# B&R Automation Studio project TD52 (part 63)

```c
  for (i = 0; i < 13; i++) {
    rtb_y_map_new[i] = Gen2_ref_DWork->y_map[i];
  }

  /* End of MATLAB Function: '<S716>/MATLAB Function' */

  /* Switch: '<S636>/Switch6' incorporates:
   *  Constant: '<S636>/Constant2'
   *  Logic: '<S636>/Logical Operator2'
   */
  if (Gen2_ref_B->BusInput3.SpeedCtrl.bKF_GS_xdist1 &&
      Gen2_ref_B->BusInput3.SpeedCtrl.bKF_act) {
    /* Gain: '<S636>/Gain2' */
    rtb_Gain1_o = rtb_Gain3;

    /* S-Function (sfix_look1_dyn): '<S636>/gain scheduling x_dist1' */
    /* Dynamic Look-Up Table Block: '<S636>/gain scheduling x_dist1'
     * Input0  Data Type:  Floating Point real_T
     * Input1  Data Type:  Floating Point real_T
     * Input2  Data Type:  Floating Point real_T
     * Output0 Data Type:  Floating Point real_T
     * Lookup Method: Linear_Endpoint
     *
     */
    LookUp_real_T_real_T( &(rtb_gainschedulingx_dist1), &rtb_y_map_new[0],
                         rtb_Gain1_o,
                         &Gen2_ref_B->BusInput3.SpeedCtrl.refPoint_KF_x_dist1_x
                         [0], 12U, inst);
    rtb_Gain1_o = rtb_gainschedulingx_dist1;
  } else {
    rtb_Gain1_o = 0.0;
  }

  /* SignalConversion generated from: '<S627>/ SFunction ' incorporates:
   *  MATLAB Function: '<S431>/LQR Controller 3states'
   *  Sum: '<S641>/Sum2'
   *  Sum: '<S641>/Sum6'
   */
  rtb_TmpSignalConversionAtSFun_g[0] = rtb_Sum1_l;
  rtb_TmpSignalConversionAtSFun_g[1] = rtb_Sum2_a_tmp;
  rtb_TmpSignalConversionAtSFun_g[2] = rtb_Sum6_o_tmp;

  /* SignalConversion generated from: '<S627>/ SFunction ' incorporates:
   *  MATLAB Function: '<S431>/LQR Controller 3states'
   */
  rtb_Divide_ab[0] = rtb_Sum2_a_tmp;
  rtb_Divide_ab[1] = rtb_Sum6_o_tmp;
  rtb_Divide_ab[2] = rtb_Switch2_oou;
  rtb_Divide_ab[3] = rtb_Sum3_o;

  /* SignalConversion generated from: '<S627>/ SFunction ' incorporates:
   *  Gain: '<S431>/Gain1'
   *  MATLAB Function: '<S431>/LQR Controller 3states'
   */
  rtb_TmpSignalConversionAtSFun_p[0] = rtb_Gain1_f_tmp;
  rtb_TmpSignalConversionAtSFun_p[1] = rtb_Gain3;
  rtb_TmpSignalConversionAtSFun_p[2] = Gen2_ref_B->Filter_bd.Switch;

  /* SignalConversion generated from: '<S627>/ SFunction ' incorporates:
   *  Constant: '<S431>/Nskip_min'
   *  MATLAB Function: '<S431>/LQR Controller 3states'
   */
  rtb_Divide3_e[0] = Gen2_ref_B->BusInput3.traj.rPr_p2s_min;
  rtb_Divide3_e[1] = rtb_Switch1_k;
  rtb_Divide3_e[2] = Gen2_ref_B->BusInput3.SpeedCtrl.rDeltaZZP_min_iLQR;
  rtb_Divide3_e[3] = 0.0;

  /* SignalConversion generated from: '<S627>/ SFunction ' incorporates:
   *  MATLAB Function: '<S431>/LQR Controller 3states'
   */
  rtb_Divide3_i0[0] = Gen2_ref_B->BusInput3.traj.rPr_p2s_max;
  rtb_Divide3_i0[1] = rtb_Switch2_n5;
  rtb_Divide3_i0[2] = Gen2_ref_B->BusInput3.SpeedCtrl.rDeltaZZP_max_iLQR;
  rtb_Divide3_i0[3] = rtb_Switch9_k;

  /* SignalConversion generated from: '<S627>/ SFunction ' incorporates:
   *  Constant: '<S639>/Constant'
   *  DataTypeConversion: '<S639>/Data Type Conversion'
   *  DataTypeConversion: '<S639>/Data Type Conversion1'
   *  MATLAB Function: '<S431>/LQR Controller 3states'
   *  Product: '<S639>/Product'
   */
  rtb_TmpSignalConversionAtSFunct[0] =
    Gen2_ref_B->BusInput3.SpeedCtrl.iNiter_iLQR;
  rtb_TmpSignalConversionAtSFunct[1] = rtb_Product1_b4;
  rtb_TmpSignalConversionAtSFunct[2] = Gen2_ref_B->BusInput3.eng.Ts;
  rtb_TmpSignalConversionAtSFunct[3] = Gen2_ref_B->BusInput3.eng.rJ_Eng *
    Gen2_ref_B->BusInput3.SpeedCtrl.rFactInertiaLQR;
  rtb_TmpSignalConversionAtSFunct[4] = rtb_Product_o;
  rtb_TmpSignalConversionAtSFunct[5] = rtb_Switch_czo;
  rtb_TmpSignalConversionAtSFunct[6] = rtb_Sum2_kg;
  rtb_TmpSignalConversionAtSFunct[7] =
    Gen2_ref_B->BusInput3.SpeedCtrl.rK_it2_iLQR;
  rtb_TmpSignalConversionAtSFunct[8] = rtb_Sum1_idx_2;
  rtb_TmpSignalConversionAtSFunct[9] = rtb_kappa0;
  rtb_TmpSignalConversionAtSFunct[10] =
    Gen2_ref_B->BusInput3.SpeedCtrl.rK_slope_iLQR;
  rtb_TmpSignalConversionAtSFunct[11] =
    Gen2_ref_B->BusInput3.SpeedCtrl.rK_skip_iLQR;
  rtb_TmpSignalConversionAtSFunct[12] = Gen2_ref_B->BusInput3.eng.rNum_Cyl_Eng;
  rtb_TmpSignalConversionAtSFunct[13] =
    Gen2_ref_B->BusInput3.SpeedCtrl.rN_DB_Lambda_act;
  rtb_TmpSignalConversionAtSFunct[14] = 1.0;
  rtb_TmpSignalConversionAtSFunct[15] =
    Gen2_ref_B->BusInput3.SpeedCtrl.iNiterRediLQR;
  rtb_TmpSignalConversionAtSFunct[16] = rtb_Product1_fu;
  rtb_TmpSignalConversionAtSFunct[17] = Gen2_ref_B->BusInput3.eng.rP_Nom;
  rtb_TmpSignalConversionAtSFunct[18] = Gen2_ref_B->BusInput3.eng.rN_Nom;
  rtb_TmpSignalConversionAtSFunct[19] = Gen2_ref_B->BusInput3.traj.rPr_p2s_max;
  rtb_TmpSignalConversionAtSFunct[20] = Gen2_ref_B->BusInput3.LamLim.rLam_max;
  rtb_TmpSignalConversionAtSFunct[21] = rtb_Divide3_g;

  /* MATLAB Function: '<S431>/LQR Controller 3states' incorporates:
   *  DataTypeConversion: '<S639>/Data Type Conversion'
   *  DataTypeConversion: '<S639>/Data Type Conversion1'
   *  Delay: '<S431>/Delay'
   *  Gain: '<S431>/Gain1'
   *  Logic: '<S636>/Logical Operator1'
   *  SignalConversion generated from: '<S627>/ SFunction '
   *  Sum: '<S641>/Sum2'
   *  Sum: '<S641>/Sum6'
   *  Switch: '<S636>/Switch7'
   */
  rtb_Switch2_l = rtb_Gain1_f_tmp;
  y_map_tmp = rtb_Gain3;
  y_map_tmp_0 = Gen2_ref_B->Filter_bd.Switch;
  Gen2_ref_diag(&rtb_Product_m[0], R_2inp, inst);
  Gen2_ref_diag_i(rtb_Product_m, R, inst);
  Gen2_ref_diag_i2(rtb_Switch1_cl, Q, inst);
  for (i = 0; i < 12; i++) {
    rtb_K_LQR[i] = 0.0;
    K_2inp_aug[i] = 0.0;
  }

  delta_y = rt_roundd_snf(rtb_Product1_b4 / Gen2_ref_B->BusInput3.eng.Ts, inst);
  if (delta_y < 32768.0) {
    if (delta_y >= -32768.0) {
      Npred = (int16_T)delta_y;
    } else {
      Npred = MIN_int16_T;
    }
  } else {
    Npred = MAX_int16_T;
  }

  rtb_Product1_b4 = Gen2_ref_B->BusInput3.SpeedCtrl.rN_DB_Lambda_act *
    3.1415926535897931 / 30.0;
  rtb_TmpSignalConversionAtLoo_ht[1] = Gen2_ref_B->BusInput3.eng.rNum_Cyl_Eng;
  if (1.0 < rtb_TmpSignalConversionAtLoo_ht[1]) {
    delta_y = rtb_TmpSignalConversionAtLoo_ht[1];
  } else {
    delta_y = 1.0;
  }

  rtb_Sum2_kg = (1.0 - rtb_Divide3_g / delta_y) * rtb_Product_o;
  Gen2_ref_diag_i2(Gen2_ref_B->BusInput3.SpeedCtrl.rBd_KF, B_d, inst);
  rtb_Switch1_cl[0] = 0.0;
  rtb_Switch1_cl[1] = 0.0;
  rtb_Switch1_cl[2] = 0.0;
  Gen2_ref_diag_i2(Gen2_ref_B->BusInput3.SpeedCtrl.rR_KF, R_KF, inst);
  if (Gen2_ref_B->BusInput3.SpeedCtrl.bKF_x_dist1_AdaptON &&
      Gen2_ref_B->BusInput3.SpeedCtrl.bKF_GS_xdist1 &&
      Gen2_ref_B->TON_j.LogicalOperator3) {
    Gen2_ref_DWork->x_KF[0] = rtb_Gain1_f_tmp;
    Gen2_ref_DWork->x_KF[3] = 0.0;
    Gen2_ref_DWork->x_KF[1] = rtb_Gain3;
    Gen2_ref_DWork->x_KF[4] = 0.0;
    Gen2_ref_DWork->x_KF[2] = Gen2_ref_B->Filter_bd.Switch;
    Gen2_ref_DWork->x_KF[5] = 0.0;
  }

  if ((!Gen2_ref_DWork->P_not_empty) || rtb_bResetHlci) {
    for (i = 0; i < 9; i++) {
      Gen2_ref_DWork->P[i] = 0.0;
    }

    Gen2_ref_DWork->P_not_empty = true;
    for (i = 0; i < 36; i++) {
      Gen2_ref_DWork->P_2inp_aug[i] = 0.0;
    }

    for (i = 0; i < 100; i++) {
      Gen2_ref_DWork->u2_past[i] = rtb_Sum6_o_tmp;
    }

    Gen2_ref_DWork->count = 1.0;
    Gen2_ref_DWork->red_comp = false;
    rtb_Product_m[0] = rtb_Sum2_a_tmp;
    rtb_Product_m[1] = rtb_Sum6_o_tmp;
    rtb_Product_m[2] = rtb_Switch2_oou;
    rtb_Product_m[3] = rtb_Sum3_o;
    Gen2_ref_DWork->x_KF[0] = rtb_Gain1_f_tmp;
    Gen2_ref_DWork->x_KF[3] = 0.0;
    Gen2_ref_DWork->x_KF[1] = rtb_Gain3;
    Gen2_ref_DWork->x_KF[4] = 0.0;
    Gen2_ref_DWork->x_KF[2] = Gen2_ref_B->Filter_bd.Switch;
    Gen2_ref_DWork->x_KF[5] = 0.0;
    for (i = 0; i < 36; i++) {
      Gen2_ref_DWork->P_KF[i] = c[i];
    }

    for (i = 0; i < 18; i++) {
      rtb_K_KF_out[i] = 0.0;
    }

    rtb_err_KF[0] = 0.0;
    rtb_x_KF_out_idx_0 = rtb_Gain1_f_tmp;
    rtb_x_sp_KF_idx_0 = rtb_Sum1_l;
    rtb_err_KF[1] = 0.0;
    rtb_x_KF_out_idx_1 = rtb_Gain3;
    rtb_x_sp_KF_idx_1 = rtb_Sum2_a_tmp;
    rtb_err_KF[2] = 0.0;
    rtb_x_KF_out_idx_2 = Gen2_ref_B->Filter_bd.Switch;
    rtb_x_sp_KF_idx_2 = rtb_Sum6_o_tmp;
    rtb_u_sp_KF[0] = rtb_Sum2_a_tmp;
    rtb_u_sp_KF[1] = rtb_Sum6_o_tmp;
    Gen2_ref_state_space_d(rtb_TmpSignalConversionAtSFun_g,
      rtb_TmpSignalConversionAtSFunct, rtb_Product_o, rtb_Phi_OUT, rtb_H_OUT,
      Hd_obs, inst);
    for (i = 0; i < 3; i++) {
      rtb_err_cont[i] = 0.0;
      Phi_aug_tmp_0 = i << 2;
      K_2inp_aug[Phi_aug_tmp_0] = rtb_H_OUT[i];
      K_2inp_aug[Phi_aug_tmp_0 + 1] = rtb_H_OUT[i + 3];
      K_2inp_aug[Phi_aug_tmp_0 + 2] = rtb_H_OUT[i + 6];
      K_2inp_aug[Phi_aug_tmp_0 + 3] = rtb_H_OUT[i + 9];
    }

    for (i = 0; i < 4; i++) {
      for (Phi_aug_tmp = 0; Phi_aug_tmp < 3; Phi_aug_tmp++) {
        Phi_aug_tmp_0 = (Phi_aug_tmp << 2) + i;
        rtb_H_OUT_0[Phi_aug_tmp_0] = 0.0;
        rtb_H_OUT_0[Phi_aug_tmp_0] += Gen2_ref_DWork->P[3 * Phi_aug_tmp] *
          K_2inp_aug[i];
        rtb_H_OUT_0[Phi_aug_tmp_0] += Gen2_ref_DWork->P[3 * Phi_aug_tmp + 1] *
          K_2inp_aug[i + 4];
        rtb_H_OUT_0[Phi_aug_tmp_0] += Gen2_ref_DWork->P[3 * Phi_aug_tmp + 2] *
          K_2inp_aug[i + 8];
      }

      for (Phi_aug_tmp = 0; Phi_aug_tmp < 4; Phi_aug_tmp++) {
        rtb_H_OUT_tmp = (Phi_aug_tmp << 2) + i;
        R_0[rtb_H_OUT_tmp] = -(((rtb_H_OUT[3 * Phi_aug_tmp + 1] * rtb_H_OUT_0[i
          + 4] + rtb_H_OUT[3 * Phi_aug_tmp] * rtb_H_OUT_0[i]) + rtb_H_OUT[3 *
          Phi_aug_tmp + 2] * rtb_H_OUT_0[i + 8]) + R[rtb_H_OUT_tmp]);
      }
    }

    Gen2_ref_mldivide(R_0, K_2inp_aug, rtb_K_LQR_0, inst);
    for (i = 0; i < 4; i++) {
      for (Phi_aug_tmp = 0; Phi_aug_tmp < 3; Phi_aug_tmp++) {
        rtb_H_OUT_tmp = (Phi_aug_tmp << 2) + i;
        tmp[rtb_H_OUT_tmp] = 0.0;
        tmp[rtb_H_OUT_tmp] += Gen2_ref_DWork->P[3 * Phi_aug_tmp] * rtb_K_LQR_0[i];
        tmp[rtb_H_OUT_tmp] += Gen2_ref_DWork->P[3 * Phi_aug_tmp + 1] *
          rtb_K_LQR_0[i + 4];
        tmp[rtb_H_OUT_tmp] += Gen2_ref_DWork->P[3 * Phi_aug_tmp + 2] *
          rtb_K_LQR_0[i + 8];
      }

      for (Phi_aug_tmp = 0; Phi_aug_tmp < 3; Phi_aug_tmp++) {
        Phi_aug_tmp_0 = (Phi_aug_tmp << 2) + i;
        rtb_K_LQR[Phi_aug_tmp_0] = 0.0;
        rtb_K_LQR[Phi_aug_tmp_0] += rtb_Phi_OUT[3 * Phi_aug_tmp] * tmp[i];
        rtb_K_LQR[Phi_aug_tmp_0] += rtb_Phi_OUT[3 * Phi_aug_tmp + 1] * tmp[i + 4];
        rtb_K_LQR[Phi_aug_tmp_0] += rtb_Phi_OUT[3 * Phi_aug_tmp + 2] * tmp[i + 8];
      }
    }
  } else {
    if (Gen2_ref_DWork->red_comp) {
      rtb_Product1_fu = Gen2_ref_B->BusInput3.SpeedCtrl.iNiterRediLQR;
    } else {
      rtb_Product1_fu = Gen2_ref_B->BusInput3.SpeedCtrl.iNiter_iLQR;
    }

    Gen2_ref_state_space_d(rtb_TmpSignalConversionAtSFun_p,
      rtb_TmpSignalConversionAtSFunct, rtb_Product_o, rtb_Phi_OUT, rtb_H_OUT,
      Hd_obs, inst);
    if (Gen2_ref_B->BusInput3.SpeedCtrl.bKF_KeNskip_Obs) {
      Gen2_ref_state_space_d(rtb_TmpSignalConversionAtSFun_p,
        rtb_TmpSignalConversionAtSFunct, rtb_Sum2_kg, Phi_obs, H_aug, Hd_obs, inst);
    } else {
      Gen2_ref_state_space_d(rtb_TmpSignalConversionAtSFun_p,
        rtb_TmpSignalConversionAtSFunct, rtb_Product_o, Phi_obs, H_aug, Hd_obs, inst);
    }

    if (Gen2_ref_B->BusInput3.SpeedCtrl.bKF_use_Pg) {
      rtb_Sum4_g = rtb_Divide3_ep;
    } else {
      rtb_Sum4_g = rtb_Divide_i1;
    }

    if (Gen2_ref_B->BusInput3.SpeedCtrl.bKF_calc ||
        Gen2_ref_B->BusInput3.SpeedCtrl.bKF_act ||
        Gen2_ref_B->BusInput3.SpeedCtrl.bKF_use_states) {
      rtb_Switch_n = Gen2_ref_B->BusInput3.eng.Ts;
      for (i = 0; i < 3; i++) {
        Phi_aug[6 * i] = Phi_obs[3 * i];
        Phi_aug_tmp_0 = (i + 3) * 6;
        Phi_aug[Phi_aug_tmp_0] = B_d[3 * i] * rtb_Switch_n;
        Phi_aug_tmp = 3 * i + 1;
        Phi_aug[6 * i + 1] = Phi_obs[Phi_aug_tmp];
        Phi_aug[Phi_aug_tmp_0 + 1] = B_d[Phi_aug_tmp] * rtb_Switch_n;
        Phi_aug_tmp = 3 * i + 2;
        Phi_aug[6 * i + 2] = Phi_obs[Phi_aug_tmp];
        Phi_aug[Phi_aug_tmp_0 + 2] = B_d[Phi_aug_tmp] * rtb_Switch_n;
      }

      for (i = 0; i < 6; i++) {
        Phi_aug[6 * i + 3] = b[3 * i];
        Phi_aug[6 * i + 4] = b[3 * i + 1];
        Phi_aug[6 * i + 5] = b[3 * i + 2];
      }

      rtb_Sum5_iu = Gen2_ref_B->BusInput3.eng.rNum_Cyl_Eng;
      if (Gen2_ref_B->BusInput3.eng.rNum_Cyl_Eng < 1.0) {
        rtb_Sum5_iu = 1.0;
      }

      rtb_TmpSignalConversionAtSFun_0[0] = (1.0 - rtb_Divide3_g / rtb_Sum5_iu) *
        rtb_Product_o * Gen2_ref_B->BusInput3.eng.Ts * Gen2_ref_DWork->x_KF[1] /
        ((Gen2_ref_DWork->x_KF[2] * rtb_Sum1_idx_2 + 1.0) *
         rtb_TmpSignalConversionAtSFunct[3]);
      rtb_TmpSignalConversionAtSFun_0[1] = Gen2_ref_B->BusInput3.eng.Ts /
        rtb_Switch_czo * (Gen2_ref_DWork->Delay_DSTATE_ba[0] -
                          Gen2_ref_DWork->x_KF[1]);
      rtb_TmpSignalConversionAtSFun_0[2] = Gen2_ref_B->BusInput3.eng.Ts /
        rtb_TmpSignalConversionAtSFunct[6] * (Gen2_ref_DWork->Delay_DSTATE_ba[1]
        - Gen2_ref_DWork->x_KF[2]);
      rtb_TmpSignalConversionAtSFun_0[3] = 0.0;
      Hd_obs_0[0] = Gen2_ref_DWork->x_KF[0];
      Hd_obs_0[3] = 0.0;
      rtb_TmpSignalConversionAtSFun_0[4] = 0.0;
      Hd_obs_0[1] = Gen2_ref_DWork->x_KF[1];
      Hd_obs_0[4] = 0.0;
      rtb_TmpSignalConversionAtSFun_0[5] = 0.0;
      Hd_obs_0[2] = Gen2_ref_DWork->x_KF[2];
      Hd_obs_0[5] = 0.0;
      for (i = 0; i < 6; i++) {
        rtb_TmpSignalConversionAtSFun_1[i] = ((Phi_aug[i + 18] *
          Gen2_ref_DWork->x_KF[3] + Phi_aug[i + 24] * Gen2_ref_DWork->x_KF[4]) +
          Phi_aug[i + 30] * Gen2_ref_DWork->x_KF[5]) +
          (rtb_TmpSignalConversionAtSFun_0[i] + Hd_obs_0[i]);
      }

      Hd_obs_0[0] = Hd_obs[0] * rtb_Sum4_g;
      Hd_obs_0[3] = 0.0 * rtb_Sum4_g;
      Hd_obs_0[1] = Hd_obs[1] * rtb_Sum4_g;
      Hd_obs_0[4] = 0.0 * rtb_Sum4_g;
      Hd_obs_0[2] = Hd_obs[2] * rtb_Sum4_g;
      Hd_obs_0[5] = 0.0 * rtb_Sum4_g;
      rtb_TmpSignalConversionAtSFun_0[0] = B_d[0] * rtb_Gain1_o *
        Gen2_ref_B->BusInput3.eng.Ts;
      for (i = 0; i < 5; i++) {
        rtb_TmpSignalConversionAtSFun_0[i + 1] = 0.0;
      }

      for (i = 0; i < 6; i++) {
        x_[i] = (rtb_TmpSignalConversionAtSFun_1[i] + Hd_obs_0[i]) +
          rtb_TmpSignalConversionAtSFun_0[i];
        for (Phi_aug_tmp = 0; Phi_aug_tmp < 6; Phi_aug_tmp++) {
          Phi_aug_0[Phi_aug_tmp + 6 * i] = 0.0;
        }

        for (rtb_H_OUT_tmp = 0; rtb_H_OUT_tmp < 6; rtb_H_OUT_tmp++) {
          for (Phi_aug_tmp = 0; Phi_aug_tmp < 6; Phi_aug_tmp++) {
            Phi_aug_tmp_0 = 6 * i + Phi_aug_tmp;
            Phi_aug_0[Phi_aug_tmp_0] += Phi_aug[6 * rtb_H_OUT_tmp + Phi_aug_tmp]
              * Gen2_ref_DWork->P_KF[6 * i + rtb_H_OUT_tmp];
          }
        }
      }

      Gen2_ref_diag_i2a(Gen2_ref_B->BusInput3.SpeedCtrl.rQ_KF, Phi_aug_1, inst);
      for (i = 0; i < 6; i++) {
        for (Phi_aug_tmp = 0; Phi_aug_tmp < 6; Phi_aug_tmp++) {
          delta_y = 0.0;
          for (rtb_H_OUT_tmp = 0; rtb_H_OUT_tmp < 6; rtb_H_OUT_tmp++) {
            delta_y += Phi_aug_0[6 * rtb_H_OUT_tmp + i] * Phi_aug[6 *
              rtb_H_OUT_tmp + Phi_aug_tmp];
          }

          Phi_aug_tmp_0 = 6 * Phi_aug_tmp + i;
          P_[Phi_aug_tmp_0] = Phi_aug_1[Phi_aug_tmp_0] + delta_y;
        }
      }

      for (i = 0; i < 18; i++) {
        Phi_obs_tmp[i] = C_aug[i];
        rtb_K_KF_out[i] = d[i];
      }

      for (i = 0; i < 3; i++) {
        for (Phi_aug_tmp = 0; Phi_aug_tmp < 6; Phi_aug_tmp++) {
          k = 3 * Phi_aug_tmp + i;
          Phi_obs_tmp_0[k] = 0.0;
          for (rtb_H_OUT_tmp = 0; rtb_H_OUT_tmp < 6; rtb_H_OUT_tmp++) {
            Phi_obs_tmp_0[k] += (real_T)Phi_obs_tmp[3 * rtb_H_OUT_tmp + i] * P_
              [6 * Phi_aug_tmp + rtb_H_OUT_tmp];
          }
        }

        for (Phi_aug_tmp = 0; Phi_aug_tmp < 3; Phi_aug_tmp++) {
          delta_y = 0.0;
          for (rtb_H_OUT_tmp = 0; rtb_H_OUT_tmp < 6; rtb_H_OUT_tmp++) {
            delta_y += Phi_obs_tmp_0[3 * rtb_H_OUT_tmp + i] * rtb_K_KF_out[6 *
              Phi_aug_tmp + rtb_H_OUT_tmp];
          }

          k = 3 * Phi_aug_tmp + i;
          Phi_obs[k] = R_KF[k] + delta_y;
        }
      }

      if (fabs(Gen2_ref_det(Phi_obs, inst)) <= 2.2204460492503131E-16) {
        for (i = 0; i < 3; i++) {
          for (Phi_aug_tmp = 0; Phi_aug_tmp < 6; Phi_aug_tmp++) {
            k = 3 * Phi_aug_tmp + i;
            Phi_obs_tmp_0[k] = 0.0;
            for (rtb_H_OUT_tmp = 0; rtb_H_OUT_tmp < 6; rtb_H_OUT_tmp++) {
              Phi_obs_tmp_0[k] += (real_T)Phi_obs_tmp[3 * rtb_H_OUT_tmp + i] *
                Gen2_ref_DWork->P_KF[6 * Phi_aug_tmp + rtb_H_OUT_tmp];
            }
          }

          for (Phi_aug_tmp = 0; Phi_aug_tmp < 3; Phi_aug_tmp++) {
            delta_y = 0.0;
            for (rtb_H_OUT_tmp = 0; rtb_H_OUT_tmp < 6; rtb_H_OUT_tmp++) {
              delta_y += Phi_obs_tmp_0[3 * rtb_H_OUT_tmp + i] * rtb_K_KF_out[6 *
                Phi_aug_tmp + rtb_H_OUT_tmp];
            }

            k = 3 * Phi_aug_tmp + i;
            Phi_obs[k] = R_KF[k] + delta_y;
          }
        }
      }

      for (i = 0; i < 3; i++) {
        for (Phi_aug_tmp = 0; Phi_aug_tmp < 6; Phi_aug_tmp++) {
          Phi_aug_tmp_0 = 6 * i + Phi_aug_tmp;
          Phi_obs_tmp_0[Phi_aug_tmp_0] = 0.0;
          for (rtb_H_OUT_tmp = 0; rtb_H_OUT_tmp < 6; rtb_H_OUT_tmp++) {
            Phi_obs_tmp_0[Phi_aug_tmp_0] += P_[6 * rtb_H_OUT_tmp + Phi_aug_tmp] *
              rtb_K_KF_out[6 * i + rtb_H_OUT_tmp];
          }
        }
      }

      Gen2_ref_mrdiv(Phi_obs_tmp_0, Phi_obs, rtb_K_KF_out, inst);
      for (i = 0; i < 6; i++) {
        for (Phi_aug_tmp = 0; Phi_aug_tmp < 3; Phi_aug_tmp++) {
          k = 6 * Phi_aug_tmp + i;
          Phi_obs_tmp_0[k] = 0.0;
          Phi_obs_tmp_0[k] += Phi_obs[3 * Phi_aug_tmp] * rtb_K_KF_out[i];
          Phi_obs_tmp_0[k] += Phi_obs[3 * Phi_aug_tmp + 1] * rtb_K_KF_out[i + 6];
          Phi_obs_tmp_0[k] += Phi_obs[3 * Phi_aug_tmp + 2] * rtb_K_KF_out[i + 12];
        }

        for (Phi_aug_tmp = 0; Phi_aug_tmp < 6; Phi_aug_tmp++) {
          k = 6 * Phi_aug_tmp + i;
          Gen2_ref_DWork->P_KF[k] = P_[k] - ((Phi_obs_tmp_0[i + 6] *
            rtb_K_KF_out[Phi_aug_tmp + 6] + Phi_obs_tmp_0[i] *
            rtb_K_KF_out[Phi_aug_tmp]) + Phi_obs_tmp_0[i + 12] *
            rtb_K_KF_out[Phi_aug_tmp + 12]);
        }
      }

      for (i = 0; i < 3; i++) {
        Phi_obs_tmp_1[i] = 0.0;
        for (Phi_aug_tmp = 0; Phi_aug_tmp < 6; Phi_aug_tmp++) {
          Phi_obs_tmp_1[i] += (real_T)Phi_obs_tmp[3 * Phi_aug_tmp + i] *
            x_[Phi_aug_tmp];
        }

        rtb_err_KF[i] = (((real_T)b_a[i + 3] * rtb_Gain3 + (real_T)b_a[i] *
                          rtb_Gain1_f_tmp) + (real_T)b_a[i + 6] *
                         Gen2_ref_B->Filter_bd.Switch) - Phi_obs_tmp_1[i];
      }

      for (i = 0; i < 6; i++) {
        Gen2_ref_DWork->x_KF[i] = ((rtb_K_KF_out[i + 6] * rtb_err_KF[1] +
          rtb_K_KF_out[i] * rtb_err_KF[0]) + rtb_K_KF_out[i + 12] * rtb_err_KF[2])
          + x_[i];
      }

      rtb_x_KF_out_idx_0 = Gen2_ref_DWork->x_KF[0];
      rtb_Switch1_cl[0] = Gen2_ref_DWork->x_KF[3];
      rtb_x_KF_out_idx_1 = Gen2_ref_DWork->x_KF[1];
      rtb_Switch1_cl[1] = Gen2_ref_DWork->x_KF[4];
      rtb_x_KF_out_idx_2 = Gen2_ref_DWork->x_KF[2];
      rtb_Switch1_cl[2] = Gen2_ref_DWork->x_KF[5];
      if (Gen2_ref_B->BusInput3.SpeedCtrl.bKF_use_states ||
          Gen2_ref_B->BusInput3.SpeedCtrl.bKF_act) {
        rtb_Switch2_l = Gen2_ref_DWork->x_KF[0];
        y_map_tmp = Gen2_ref_DWork->x_KF[1];
        y_map_tmp_0 = Gen2_ref_DWork->x_KF[2];
      }

      rtb_x_sp_KF_idx_0 = rtb_Sum1_l;
      if (Gen2_ref_B->BusInput3.SpeedCtrl.bKF_constr_handling) {
        if (Gen2_ref_B->BusInput3.SpeedCtrl.bKF_Lam_dyn_SP_shift) {
          FILT_IN = Gen2_ref_DWork->x_KF[3] + rtb_Gain1_o;
          rtb_x_sp_KF_idx_2 = ((FILT_IN * rtb_TmpSignalConversionAtSFunct[3] *
                                B_d[0] + rtb_Sum2_kg * rtb_Sum2_a_tmp) -
                               rtb_Divide_i1) / (rtb_Divide_i1 * rtb_Sum1_idx_2
            - rtb_TmpSignalConversionAtSFunct[3] * rtb_Sum1_idx_2 * FILT_IN *
            B_d[0]) + Gen2_ref_DWork->x_KF[5] * rtb_TmpSignalConversionAtSFunct
            [6] * B_d[8];
        } else {
          rtb_x_sp_KF_idx_1 = Gen2_ref_DWork->x_KF[3] + rtb_Gain1_o;
          rtb_x_sp_KF_idx_2 = ((rtb_x_sp_KF_idx_1 *
                                rtb_TmpSignalConversionAtSFunct[3] * B_d[0] +
                                rtb_Sum2_kg * rtb_Sum2_a_tmp) - rtb_Divide_i1) /
            (rtb_Divide_i1 * rtb_Sum1_idx_2 - rtb_TmpSignalConversionAtSFunct[3]
             * rtb_Sum1_idx_2 * rtb_x_sp_KF_idx_1 * B_d[0]);
        }

        if (rtb_x_sp_KF_idx_2 > rtb_Switch2_n5) {
          rtb_x_sp_KF_idx_2 = rtb_Switch2_n5;
        } else if (rtb_x_sp_KF_idx_2 < rtb_Switch1_k) {
          rtb_x_sp_KF_idx_2 = rtb_Switch1_k;
        }

        if (Gen2_ref_B->BusInput3.SpeedCtrl.bKF_p2s_dyn_SP_shift) {
          rtb_x_sp_KF_idx_1 = (rtb_Divide_i1 - (Gen2_ref_DWork->x_KF[3] +
            rtb_Gain1_o) * rtb_TmpSignalConversionAtSFunct[3] * B_d[0]) *
            (rtb_x_sp_KF_idx_2 * rtb_Sum1_idx_2 + 1.0) / rtb_Sum2_kg +
            Gen2_ref_DWork->x_KF[4] * rtb_Switch_czo * B_d[4];
        } else if ((rtb_Divide3_g > 0.0) &&
                   (!Gen2_ref_B->BusInput3.SpeedCtrl.bKF_constr_handlLR)) {
          rtb_x_sp_KF_idx_1 = rtb_Sum2_a_tmp;
        } else {
          rtb_x_sp_KF_idx_1 = (rtb_Divide_i1 - (Gen2_ref_DWork->x_KF[3] +
            rtb_Gain1_o) * rtb_TmpSignalConversionAtSFunct[3] * B_d[0]) *
            (rtb_x_sp_KF_idx_2 * rtb_Sum1_idx_2 + 1.0) / rtb_Sum2_kg;
        }
      } else {
        if (Gen2_ref_B->BusInput3.SpeedCtrl.bKF_p2s_dyn_SP_shift) {
          rtb_x_sp_KF_idx_1 = Gen2_ref_DWork->x_KF[4] * rtb_Switch_czo * B_d[4]
            + rtb_Sum2_a_tmp;
        } else {
          rtb_x_sp_KF_idx_1 = rtb_Sum2_a_tmp;
        }

        if (Gen2_ref_B->BusInput3.SpeedCtrl.bKF_Lam_dyn_SP_shift) {
          rtb_x_sp_KF_idx_2 = (((Gen2_ref_DWork->x_KF[3] + rtb_Gain1_o) *
                                rtb_TmpSignalConversionAtSFunct[3] * B_d[0] +
                                rtb_Sum2_kg * rtb_Sum2_a_tmp) - rtb_Divide_i1) /
            (rtb_Divide_i1 * rtb_Sum1_idx_2 - rtb_TmpSignalConversionAtSFunct[3]
             * rtb_Sum1_idx_2 * (Gen2_ref_DWork->x_KF[3] + rtb_Gain1_o) * B_d[0])
            + Gen2_ref_DWork->x_KF[5] * rtb_TmpSignalConversionAtSFunct[6] *
            B_d[8];
        } else {
          rtb_x_sp_KF_idx_2 = (((Gen2_ref_DWork->x_KF[3] + rtb_Gain1_o) *
                                rtb_TmpSignalConversionAtSFunct[3] * B_d[0] +
                                rtb_Sum2_kg * rtb_Sum2_a_tmp) - rtb_Divide_i1) /
            (rtb_Divide_i1 * rtb_Sum1_idx_2 - rtb_TmpSignalConversionAtSFunct[3]
             * rtb_Sum1_idx_2 * (Gen2_ref_DWork->x_KF[3] + rtb_Gain1_o) * B_d[0]);
        }
      }

      rtb_u_sp_KF[0] = rtb_x_sp_KF_idx_1;
      rtb_u_sp_KF[1] = rtb_x_sp_KF_idx_2;
    } else {
      rtb_err_KF[0] = 0.0;
      rtb_x_KF_out_idx_0 = rtb_Gain1_f_tmp * 0.0;
      rtb_x_sp_KF_idx_0 = 0.0;
      rtb_err_KF[1] = 0.0;
      rtb_x_KF_out_idx_1 = rtb_Gain3 * 0.0;
      rtb_x_sp_KF_idx_1 = 0.0;
      rtb_err_KF[2] = 0.0;
      rtb_x_KF_out_idx_2 = Gen2_ref_B->Filter_bd.Switch * 0.0;
      rtb_x_sp_KF_idx_2 = 0.0;
      rtb_u_sp_KF[0] = 0.0;
      rtb_u_sp_KF[1] = 0.0;
      for (i = 0; i < 18; i++) {
        rtb_K_KF_out[i] = 0.0;
      }
    }

    rtb_err_cont[0] = rtb_Sum1_l - rtb_Switch2_l;
    rtb_err_cont[1] = rtb_Sum2_a_tmp - y_map_tmp;
    rtb_err_cont[2] = rtb_Sum6_o_tmp - y_map_tmp_0;
    if (Gen2_ref_B->BusInput3.SpeedCtrl.bKF_act) {
      rtb_Switch_n = Gen2_ref_B->BusInput3.eng.Ts;
      for (i = 0; i < 3; i++) {
        Phi_aug[6 * i] = rtb_Phi_OUT[3 * i];
        Phi_aug_tmp_0 = (i + 3) * 6;
        Phi_aug[Phi_aug_tmp_0] = B_d[3 * i] * rtb_Switch_n;
        Phi_aug_tmp = 3 * i + 1;
        Phi_aug[6 * i + 1] = rtb_Phi_OUT[Phi_aug_tmp];
        Phi_aug[Phi_aug_tmp_0 + 1] = B_d[Phi_aug_tmp] * rtb_Switch_n;
        Phi_aug_tmp = 3 * i + 2;
        Phi_aug[6 * i + 2] = rtb_Phi_OUT[Phi_aug_tmp];
        Phi_aug[Phi_aug_tmp_0 + 2] = B_d[Phi_aug_tmp] * rtb_Switch_n;
      }

      for (i = 0; i < 6; i++) {
        Phi_aug[6 * i + 3] = b[3 * i];
        Phi_aug[6 * i + 4] = b[3 * i + 1];
        Phi_aug[6 * i + 5] = b[3 * i + 2];
      }

      for (i = 0; i < 2; i++) {
        H_aug[6 * i] = rtb_H_OUT[3 * i];
        H_aug[6 * i + 3] = 0.0;
        H_aug[6 * i + 1] = rtb_H_OUT[3 * i + 1];
        H_aug[6 * i + 4] = 0.0;
        H_aug[6 * i + 2] = rtb_H_OUT[3 * i + 2];
        H_aug[6 * i + 5] = 0.0;
      }

      for (i = 0; i < 3; i++) {
        P_[6 * i] = Q[3 * i];
        Phi_aug_tmp_0 = (i + 3) * 6;
        P_[Phi_aug_tmp_0] = 0.0;
        P_[6 * i + 1] = Q[3 * i + 1];
        P_[Phi_aug_tmp_0 + 1] = 0.0;
        P_[6 * i + 2] = Q[3 * i + 2];
        P_[Phi_aug_tmp_0 + 2] = 0.0;
      }

      for (i = 0; i < 6; i++) {
        P_[6 * i + 3] = 0.0;
        P_[6 * i + 4] = 0.0;
        P_[6 * i + 5] = 0.0;
      }

      if (0 <= (int32_T)rtb_Product1_fu - 1) {
        for (i = 0; i < 6; i++) {
          Phi_aug_tmp_0 = i << 1;
          rtb_K_LQR[Phi_aug_tmp_0] = H_aug[i];
          rtb_K_LQR[Phi_aug_tmp_0 + 1] = H_aug[i + 6];
        }
      }

      for (k = 0; k < (int32_T)rtb_Product1_fu; k++) {
        for (i = 0; i < 2; i++) {
          for (Phi_aug_tmp = 0; Phi_aug_tmp < 6; Phi_aug_tmp++) {
            Phi_aug_tmp_0 = (Phi_aug_tmp << 1) + i;
            rtb_K_LQR_0[Phi_aug_tmp_0] = 0.0;
            for (rtb_H_OUT_tmp = 0; rtb_H_OUT_tmp < 6; rtb_H_OUT_tmp++) {
              rtb_K_LQR_0[Phi_aug_tmp_0] += rtb_K_LQR[(rtb_H_OUT_tmp << 1) + i] *
                Gen2_ref_DWork->P_2inp_aug[6 * Phi_aug_tmp + rtb_H_OUT_tmp];
            }
          }

          for (Phi_aug_tmp = 0; Phi_aug_tmp < 2; Phi_aug_tmp++) {
            delta_y = 0.0;
            for (rtb_H_OUT_tmp = 0; rtb_H_OUT_tmp < 6; rtb_H_OUT_tmp++) {
              delta_y += rtb_K_LQR_0[(rtb_H_OUT_tmp << 1) + i] * H_aug[6 *
                Phi_aug_tmp + rtb_H_OUT_tmp];
            }

            rtb_H_OUT_tmp = (Phi_aug_tmp << 1) + i;
            rtb_Product_m[rtb_H_OUT_tmp] = -(R_2inp[rtb_H_OUT_tmp] + delta_y);
          }
        }

        Gen2_ref_mldivide_j(rtb_Product_m, rtb_K_LQR, rtb_K_LQR_0, inst);
        for (i = 0; i < 2; i++) {
          for (Phi_aug_tmp = 0; Phi_aug_tmp < 6; Phi_aug_tmp++) {
            rtb_H_OUT_tmp = (Phi_aug_tmp << 1) + i;
            tmp[rtb_H_OUT_tmp] = 0.0;
            for (Phi_aug_tmp_0 = 0; Phi_aug_tmp_0 < 6; Phi_aug_tmp_0++) {
              tmp[rtb_H_OUT_tmp] += rtb_K_LQR_0[(Phi_aug_tmp_0 << 1) + i] *
                Gen2_ref_DWork->P_2inp_aug[6 * Phi_aug_tmp + Phi_aug_tmp_0];
            }
          }

          for (Phi_aug_tmp = 0; Phi_aug_tmp < 6; Phi_aug_tmp++) {
            Phi_aug_tmp_0 = (Phi_aug_tmp << 1) + i;
            K_2inp_aug[Phi_aug_tmp_0] = 0.0;
            for (rtb_H_OUT_tmp = 0; rtb_H_OUT_tmp < 6; rtb_H_OUT_tmp++) {
              K_2inp_aug[Phi_aug_tmp_0] += tmp[(rtb_H_OUT_tmp << 1) + i] *
                Phi_aug[6 * Phi_aug_tmp + rtb_H_OUT_tmp];
            }
          }
        }

        for (i = 0; i < 6; i++) {
          rtb_H_OUT_0[i] = 0.0;
          Phi_aug_tmp_0 = i << 1;
          rtb_Sum2_kg = K_2inp_aug[Phi_aug_tmp_0];
          rtb_H_OUT_0[i] += rtb_Sum2_kg * R_2inp[0];
          rtb_Switch_czo = K_2inp_aug[Phi_aug_tmp_0 + 1];
          rtb_H_OUT_0[i] += rtb_Switch_czo * R_2inp[1];
          rtb_H_OUT_0[i + 6] = 0.0;
          rtb_H_OUT_0[i + 6] += rtb_Sum2_kg * R_2inp[2];
          rtb_H_OUT_0[i + 6] += rtb_Switch_czo * R_2inp[3];
          for (Phi_aug_tmp = 0; Phi_aug_tmp < 6; Phi_aug_tmp++) {
            rtb_H_OUT_tmp = 6 * Phi_aug_tmp + i;
            P_2inp_aug_tmp[rtb_H_OUT_tmp] = 0.0;
            Phi_aug_tmp_0 = Phi_aug_tmp << 1;
            P_2inp_aug_tmp[rtb_H_OUT_tmp] += K_2inp_aug[Phi_aug_tmp_0] * H_aug[i];
            P_2inp_aug_tmp[rtb_H_OUT_tmp] += K_2inp_aug[Phi_aug_tmp_0 + 1] *
              H_aug[i + 6];
            Phi_aug_0[Phi_aug_tmp + 6 * i] = Phi_aug[rtb_H_OUT_tmp] +
              P_2inp_aug_tmp[rtb_H_OUT_tmp];
          }
        }

        for (i = 0; i < 6; i++) {
          for (Phi_aug_tmp = 0; Phi_aug_tmp < 6; Phi_aug_tmp++) {
            Phi_aug_tmp_0 = 6 * Phi_aug_tmp + i;
            Phi_aug_1[Phi_aug_tmp_0] = 0.0;
            for (rtb_H_OUT_tmp = 0; rtb_H_OUT_tmp < 6; rtb_H_OUT_tmp++) {
              Phi_aug_1[Phi_aug_tmp_0] += Phi_aug_0[6 * rtb_H_OUT_tmp + i] *
                Gen2_ref_DWork->P_2inp_aug[6 * Phi_aug_tmp + rtb_H_OUT_tmp];
            }
          }
        }

        for (i = 0; i < 36; i++) {
          Phi_aug_0[i] = Phi_aug[i] + P_2inp_aug_tmp[i];
        }

        for (i = 0; i < 6; i++) {
          for (Phi_aug_tmp = 0; Phi_aug_tmp < 6; Phi_aug_tmp++) {
            Phi_aug_tmp_0 = Phi_aug_tmp << 1;
            rtb_K_LQR_tmp = 6 * Phi_aug_tmp + i;
            P_2inp_aug_tmp[rtb_K_LQR_tmp] = (K_2inp_aug[Phi_aug_tmp_0 + 1] *
              rtb_H_OUT_0[i + 6] + K_2inp_aug[Phi_aug_tmp_0] * rtb_H_OUT_0[i]) +
              P_[rtb_K_LQR_tmp];
            Phi_aug_2[rtb_K_LQR_tmp] = 0.0;
            for (rtb_H_OUT_tmp = 0; rtb_H_OUT_tmp < 6; rtb_H_OUT_tmp++) {
              Phi_aug_2[rtb_K_LQR_tmp] += Phi_aug_1[6 * rtb_H_OUT_tmp + i] *
                Phi_aug_0[6 * Phi_aug_tmp + rtb_H_OUT_tmp];
            }
          }
        }

        for (i = 0; i < 36; i++) {
          Gen2_ref_DWork->P_2inp_aug[i] = P_2inp_aug_tmp[i] + Phi_aug_2[i];
        }
      }

      for (i = 0; i < 3; i++) {
        Phi_aug_tmp_0 = i << 2;
        rtb_H_OUT_tmp = i << 1;
        rtb_K_LQR[Phi_aug_tmp_0] = K_2inp_aug[rtb_H_OUT_tmp];
        rtb_K_LQR[Phi_aug_tmp_0 + 2] = 0.0;
        rtb_K_LQR[Phi_aug_tmp_0 + 1] = K_2inp_aug[rtb_H_OUT_tmp + 1];
        rtb_K_LQR[Phi_aug_tmp_0 + 3] = 0.0;
        Gen2_ref_DWork->P[3 * i] = Gen2_ref_DWork->P_2inp_aug[6 * i];
        Gen2_ref_DWork->P[3 * i + 1] = Gen2_ref_DWork->P_2inp_aug[6 * i + 1];
        Gen2_ref_DWork->P[3 * i + 2] = Gen2_ref_DWork->P_2inp_aug[6 * i + 2];
      }
    } else {
      if (0 <= (int32_T)rtb_Product1_fu - 1) {
        for (i = 0; i < 3; i++) {
          rtb_H_OUT_tmp = i << 2;
          rtb_H_OUT_0[rtb_H_OUT_tmp] = rtb_H_OUT[i];
          rtb_H_OUT_0[rtb_H_OUT_tmp + 1] = rtb_H_OUT[i + 3];
          rtb_H_OUT_0[rtb_H_OUT_tmp + 2] = rtb_H_OUT[i + 6];
          rtb_H_OUT_0[rtb_H_OUT_tmp + 3] = rtb_H_OUT[i + 9];
        }
      }

      for (k = 0; k < (int32_T)rtb_Product1_fu; k++) {
        for (i = 0; i < 4; i++) {
          for (Phi_aug_tmp = 0; Phi_aug_tmp < 3; Phi_aug_tmp++) {
            rtb_H_OUT_tmp = (Phi_aug_tmp << 2) + i;
            rtb_K_LQR[rtb_H_OUT_tmp] = 0.0;
            rtb_K_LQR[rtb_H_OUT_tmp] += rtb_H_OUT[3 * i] * Gen2_ref_DWork->P[3 *
              Phi_aug_tmp];
            rtb_K_LQR[rtb_H_OUT_tmp] += rtb_H_OUT[3 * i + 1] * Gen2_ref_DWork->
              P[3 * Phi_aug_tmp + 1];
            rtb_K_LQR[rtb_H_OUT_tmp] += rtb_H_OUT[3 * i + 2] * Gen2_ref_DWork->
              P[3 * Phi_aug_tmp + 2];
          }

          for (Phi_aug_tmp = 0; Phi_aug_tmp < 4; Phi_aug_tmp++) {
            rtb_H_OUT_tmp = (Phi_aug_tmp << 2) + i;
            R_0[rtb_H_OUT_tmp] = -(((rtb_H_OUT[3 * Phi_aug_tmp + 1] *
              rtb_K_LQR[i + 4] + rtb_H_OUT[3 * Phi_aug_tmp] * rtb_K_LQR[i]) +
              rtb_H_OUT[3 * Phi_aug_tmp + 2] * rtb_K_LQR[i + 8]) +
              R[rtb_H_OUT_tmp]);
          }
        }

        Gen2_ref_mldivide(R_0, rtb_H_OUT_0, rtb_K_LQR_0, inst);
        for (i = 0; i < 4; i++) {
          for (Phi_aug_tmp = 0; Phi_aug_tmp < 3; Phi_aug_tmp++) {
            rtb_H_OUT_tmp = (Phi_aug_tmp << 2) + i;
            tmp[rtb_H_OUT_tmp] = 0.0;
            tmp[rtb_H_OUT_tmp] += Gen2_ref_DWork->P[3 * Phi_aug_tmp] *
              rtb_K_LQR_0[i];
            tmp[rtb_H_OUT_tmp] += Gen2_ref_DWork->P[3 * Phi_aug_tmp + 1] *
              rtb_K_LQR_0[i + 4];
            tmp[rtb_H_OUT_tmp] += Gen2_ref_DWork->P[3 * Phi_aug_tmp + 2] *
              rtb_K_LQR_0[i + 8];
          }

          for (Phi_aug_tmp = 0; Phi_aug_tmp < 3; Phi_aug_tmp++) {
            Phi_aug_tmp_0 = (Phi_aug_tmp << 2) + i;
            rtb_K_LQR[Phi_aug_tmp_0] = 0.0;
            rtb_K_LQR[Phi_aug_tmp_0] += rtb_Phi_OUT[3 * Phi_aug_tmp] * tmp[i];
            rtb_K_LQR[Phi_aug_tmp_0] += rtb_Phi_OUT[3 * Phi_aug_tmp + 1] * tmp[i
              + 4];
            rtb_K_LQR[Phi_aug_tmp_0] += rtb_Phi_OUT[3 * Phi_aug_tmp + 2] * tmp[i
              + 8];
          }
        }

        for (i = 0; i < 3; i++) {
          for (Phi_aug_tmp = 0; Phi_aug_tmp < 3; Phi_aug_tmp++) {
            rtb_H_OUT_tmp = 3 * Phi_aug_tmp + i;
            R_KF[rtb_H_OUT_tmp] = 0.0;
            Phi_aug_tmp_0 = Phi_aug_tmp << 2;
            R_KF[rtb_H_OUT_tmp] += rtb_K_LQR[Phi_aug_tmp_0] * rtb_H_OUT[i];
            R_KF[rtb_H_OUT_tmp] += rtb_K_LQR[Phi_aug_tmp_0 + 1] * rtb_H_OUT[i +
              3];
            R_KF[rtb_H_OUT_tmp] += rtb_K_LQR[Phi_aug_tmp_0 + 2] * rtb_H_OUT[i +
              6];
            R_KF[rtb_H_OUT_tmp] += rtb_K_LQR[Phi_aug_tmp_0 + 3] * rtb_H_OUT[i +
              9];
          }

          for (Phi_aug_tmp = 0; Phi_aug_tmp < 4; Phi_aug_tmp++) {
            Phi_aug_tmp_0 = 3 * Phi_aug_tmp + i;
            rtb_K_LQR_0[Phi_aug_tmp_0] = 0.0;
            rtb_H_OUT_tmp = i << 2;
            rtb_K_LQR_tmp = Phi_aug_tmp << 2;
            rtb_K_LQR_0[Phi_aug_tmp_0] += rtb_K_LQR[rtb_H_OUT_tmp] *
              R[rtb_K_LQR_tmp];
            rtb_K_LQR_0[Phi_aug_tmp_0] += rtb_K_LQR[rtb_H_OUT_tmp + 1] *
              R[rtb_K_LQR_tmp + 1];
            rtb_K_LQR_0[Phi_aug_tmp_0] += rtb_K_LQR[rtb_H_OUT_tmp + 2] *
              R[rtb_K_LQR_tmp + 2];
            rtb_K_LQR_0[Phi_aug_tmp_0] += rtb_K_LQR[rtb_H_OUT_tmp + 3] *
              R[rtb_K_LQR_tmp + 3];
          }

          Phi_obs[3 * i] = rtb_Phi_OUT[i] + R_KF[i];
          Phi_obs[3 * i + 1] = rtb_Phi_OUT[i + 3] + R_KF[i + 3];
          Phi_obs[3 * i + 2] = rtb_Phi_OUT[i + 6] + R_KF[i + 6];
        }

        for (i = 0; i < 3; i++) {
          for (Phi_aug_tmp = 0; Phi_aug_tmp < 3; Phi_aug_tmp++) {
            rtb_H_OUT_tmp = 3 * Phi_aug_tmp + i;
            rtb_Phi_OUT_0[rtb_H_OUT_tmp] = 0.0;
            rtb_Phi_OUT_0[rtb_H_OUT_tmp] += Gen2_ref_DWork->P[3 * Phi_aug_tmp] *
              Phi_obs[i];
            rtb_Phi_OUT_0[rtb_H_OUT_tmp] += Gen2_ref_DWork->P[3 * Phi_aug_tmp +
              1] * Phi_obs[i + 3];
            rtb_Phi_OUT_0[rtb_H_OUT_tmp] += Gen2_ref_DWork->P[3 * Phi_aug_tmp +
              2] * Phi_obs[i + 6];
          }
        }

        for (i = 0; i < 9; i++) {
          Phi_obs[i] = rtb_Phi_OUT[i] + R_KF[i];
        }

        for (i = 0; i < 3; i++) {
          for (Phi_aug_tmp = 0; Phi_aug_tmp < 3; Phi_aug_tmp++) {
            rtb_H_OUT_tmp = Phi_aug_tmp << 2;
            Phi_aug_tmp_0 = 3 * Phi_aug_tmp + i;
            R_KF[Phi_aug_tmp_0] = (((rtb_K_LQR[rtb_H_OUT_tmp + 1] *
              rtb_K_LQR_0[i + 3] + rtb_K_LQR[rtb_H_OUT_tmp] * rtb_K_LQR_0[i]) +
              rtb_K_LQR[rtb_H_OUT_tmp + 2] * rtb_K_LQR_0[i + 6]) +
              rtb_K_LQR[rtb_H_OUT_tmp + 3] * rtb_K_LQR_0[i + 9]) +
              Q[Phi_aug_tmp_0];
            rtb_Phi_OUT_1[Phi_aug_tmp_0] = 0.0;
            rtb_Phi_OUT_1[Phi_aug_tmp_0] += Phi_obs[3 * Phi_aug_tmp] *
              rtb_Phi_OUT_0[i];
            rtb_Phi_OUT_1[Phi_aug_tmp_0] += Phi_obs[3 * Phi_aug_tmp + 1] *
              rtb_Phi_OUT_0[i + 3];
            rtb_Phi_OUT_1[Phi_aug_tmp_0] += Phi_obs[3 * Phi_aug_tmp + 2] *
              rtb_Phi_OUT_0[i + 6];
          }
        }

        for (i = 0; i < 9; i++) {
          Gen2_ref_DWork->P[i] = R_KF[i] + rtb_Phi_OUT_1[i];
        }
      }
    }

    rtb_TmpSignalConversionAtSFun_0[0] = rtb_x_sp_KF_idx_0;
    rtb_TmpSignalConversionAtSFun_0[3] = 0.0;
    rtb_TmpSignalConversionAtSFun_1[0] = rtb_Switch2_l;
    rtb_TmpSignalConversionAtSFun_1[3] = 0.0;
    rtb_TmpSignalConversionAtSFun_0[1] = rtb_x_sp_KF_idx_1;
    rtb_TmpSignalConversionAtSFun_0[4] = 0.0;
    rtb_TmpSignalConversionAtSFun_1[1] = y_map_tmp;
    rtb_TmpSignalConversionAtSFun_1[4] = 0.0;
    rtb_TmpSignalConversionAtSFun_0[2] = rtb_x_sp_KF_idx_2;
    rtb_TmpSignalConversionAtSFun_0[5] = 0.0;
    rtb_TmpSignalConversionAtSFun_1[2] = y_map_tmp_0;
    rtb_TmpSignalConversionAtSFun_1[5] = 0.0;
    for (i = 0; i < 6; i++) {
      Hd_obs_0[i] = rtb_TmpSignalConversionAtSFun_0[i] -
        rtb_TmpSignalConversionAtSFun_1[i];
    }

    for (i = 0; i < 2; i++) {
      delta_y = 0.0;
      for (Phi_aug_tmp = 0; Phi_aug_tmp < 6; Phi_aug_tmp++) {
        delta_y += K_2inp_aug[(Phi_aug_tmp << 1) + i] * Hd_obs_0[Phi_aug_tmp];
      }

      R_2inp[i] = rtb_u_sp_KF[i] - delta_y;
    }

    R_2inp[2] = 0.0;
    R_2inp[3] = 0.0;
    if (Gen2_ref_B->BusInput3.SpeedCtrl.bKF_act) {
      for (i = 0; i < 4; i++) {
        rtb_Product_m[i] = R_2inp[i];
      }

      for (i = 0; i < 3; i++) {
        Phi_aug_tmp = i << 2;
        k = i << 1;
        H_aug[Phi_aug_tmp] = K_2inp_aug[k];
        H_aug[Phi_aug_tmp + 2] = 0.0;
        H_aug[Phi_aug_tmp + 1] = K_2inp_aug[k + 1];
        H_aug[Phi_aug_tmp + 3] = 0.0;
      }

      R_2inp[0] = rtb_u_sp_KF[0];
      R_2inp[1] = rtb_u_sp_KF[1];
      R_2inp[2] = 0.0;
      R_2inp[3] = 0.0;
      Hd_obs[0] = rtb_x_sp_KF_idx_0;
      Hd_obs[1] = rtb_x_sp_KF_idx_1;
      Hd_obs[2] = rtb_x_sp_KF_idx_2;
    } else {
      for (i = 0; i < 4; i++) {
        rtb_Product_m[i] = rtb_Divide_ab[i] - ((rtb_K_LQR[i + 4] * rtb_err_cont
          [1] + rtb_K_LQR[i] * rtb_err_cont[0]) + rtb_K_LQR[i + 8] *
          rtb_err_cont[2]);
      }

      for (i = 0; i < 12; i++) {
        H_aug[i] = rtb_K_LQR[i];
      }

      R_2inp[0] = rtb_Sum2_a_tmp;
      R_2inp[1] = rtb_Sum6_o_tmp;
      R_2inp[2] = rtb_Switch2_oou;
      R_2inp[3] = rtb_Sum3_o;
      Hd_obs[0] = rtb_Sum1_l;
      Hd_obs[1] = rtb_Sum2_a_tmp;
      Hd_obs[2] = rtb_Sum6_o_tmp;
    }

    for (i = 0; i < 100; i++) {
      u_lambda_past[i] = 0.0;
    }

    for (k = 1; k - 1 < Npred; k++) {
      i = Npred + 1;
      if (Npred + 1 > 32767) {
        i = 32767;
      }

      delta_y = rt_roundd_snf(Gen2_ref_DWork->count - (real_T)i, inst);
      if (delta_y < 32768.0) {
        if (delta_y >= -32768.0) {
          tmp_0 = (int16_T)delta_y;
        } else {
          tmp_0 = MIN_int16_T;
        }
      } else {
        tmp_0 = MAX_int16_T;
      }

      i = tmp_0 + (int16_T)k;
      if (i > 32767) {
        i = 32767;
      } else if (i < -32768) {
        i = -32768;
      }

      if (i < 1) {
        i = Npred + 1;
        if (Npred + 1 > 32767) {
          i = 32767;
        }

        delta_y = rt_roundd_snf((real_T)i - Gen2_ref_DWork->count, inst);
        if (delta_y < 32768.0) {
          if (delta_y >= -32768.0) {
            tmp_0 = (int16_T)delta_y;
          } else {
            tmp_0 = MIN_int16_T;
          }
        } else {
          tmp_0 = MAX_int16_T;
        }

        i = 100 - tmp_0;
        if (delta_y < 32768.0) {
          if (delta_y >= -32768.0) {
            tmp_0 = (int16_T)delta_y;
          } else {
            tmp_0 = MIN_int16_T;
          }
        } else {
          tmp_0 = MAX_int16_T;
        }

        if (100 - tmp_0 > 32767) {
          i = 32767;
        }

        i += (int16_T)k;
        if (i > 32767) {
          i = 32767;
        } else if (i < -32768) {
          i = -32768;
        }

        u_lambda_past[(int16_T)k - 1] = Gen2_ref_DWork->u2_past[i - 1];
      } else {
        i = Npred + 1;
        if (Npred + 1 > 32767) {
          i = 32767;
        }

        delta_y = rt_roundd_snf(Gen2_ref_DWork->count - (real_T)i, inst);
        if (delta_y < 32768.0) {
          if (delta_y >= -32768.0) {
            tmp_0 = (int16_T)delta_y;
          } else {
            tmp_0 = MIN_int16_T;
          }
        } else {
          tmp_0 = MAX_int16_T;
        }

        i = tmp_0 + (int16_T)k;
        if (i > 32767) {
          i = 32767;
        } else if (i < -32768) {
          i = -32768;
        }

        u_lambda_past[(int16_T)k - 1] = Gen2_ref_DWork->u2_past[i - 1];
      }
    }

    rtb_TmpSignalConversionAtSFun_g[0] = rtb_Switch2_l;
    rtb_TmpSignalConversionAtSFun_g[1] = y_map_tmp;
    rtb_TmpSignalConversionAtSFun_g[2] = y_map_tmp_0;
    if (!Gen2_ref_B->BusInput3.SpeedCtrl.bPredFB_usePg) {
      rtb_Divide3_ep = rtb_Divide_i1;
    }

    Gen2_ref_integrate_model(rtb_TmpSignalConversionAtSFun_g, H_aug,
      u_lambda_past, rtb_Divide3_ep, rtb_Switch1_cl, B_d, rtb_Gain1_o, R_2inp,
      Hd_obs, Npred, rtb_Divide3_e, rtb_Divide3_i0,
      rtb_TmpSignalConversionAtSFunct, inst);
    if (rtb_Product1_b4 > 0.5) {
      rtb_Product1_fu = Hd_obs[0] - rtb_TmpSignalConversionAtSFun_g[0];
      if (rtb_Product1_fu > 0.0) {
        u0 = rtb_Product1_fu - rtb_Product1_b4;
        if (u0 >= 0.0) {
          Hd_obs[0] = u0;
        } else {
          Hd_obs[0] = 0.0;
        }
      } else {
        u0 = rtb_Product1_fu + rtb_Product1_b4;
        if (u0 <= 0.0) {
          Hd_obs[0] = u0;
        } else {
          Hd_obs[0] = 0.0;
        }
      }

      rtb_Product_m[1] = R_2inp[1] - (((Hd_obs[1] -
        rtb_TmpSignalConversionAtSFun_g[1]) * H_aug[5] + Hd_obs[0] * H_aug[1]) +
        (Hd_obs[2] - rtb_TmpSignalConversionAtSFun_g[2]) * H_aug[9]);
    } else {
      rtb_Product_m[1] = R_2inp[1] - (((Hd_obs[0] -
        rtb_TmpSignalConversionAtSFun_g[0]) * H_aug[1] + (Hd_obs[1] -
        rtb_TmpSignalConversionAtSFun_g[1]) * H_aug[5]) + (Hd_obs[2] -
        rtb_TmpSignalConversionAtSFun_g[2]) * H_aug[9]);
    }

    rtb_Product1_b4 = rtb_Product_m[0];
    if (rtb_Product_m[0] > Gen2_ref_B->BusInput3.traj.rPr_p2s_max) {
      rtb_Product1_b4 = Gen2_ref_B->BusInput3.traj.rPr_p2s_max;
    } else if (rtb_Product_m[0] < Gen2_ref_B->BusInput3.traj.rPr_p2s_min) {
      rtb_Product1_b4 = Gen2_ref_B->BusInput3.traj.rPr_p2s_min;
    }

    rtb_Product_m[0] = rtb_Product1_b4;
    rtb_Product1_b4 = rtb_Product_m[1];
    if (rtb_Product_m[1] > rtb_Switch2_n5) {
      rtb_Product1_b4 = rtb_Switch2_n5;
    } else if (rtb_Product_m[1] < rtb_Switch1_k) {
      rtb_Product1_b4 = rtb_Switch1_k;
    }

    rtb_Product_m[1] = rtb_Product1_b4;
    rtb_Product1_b4 = rtb_Product_m[2];
    if (rtb_Product_m[2] > Gen2_ref_B->BusInput3.SpeedCtrl.rDeltaZZP_max_iLQR) {
      rtb_Product1_b4 = Gen2_ref_B->BusInput3.SpeedCtrl.rDeltaZZP_max_iLQR;
    } else if (rtb_Product_m[2] <
               Gen2_ref_B->BusInput3.SpeedCtrl.rDeltaZZP_min_iLQR) {
      rtb_Product1_b4 = Gen2_ref_B->BusInput3.SpeedCtrl.rDeltaZZP_min_iLQR;
    }

    rtb_Product_m[2] = rtb_Product1_b4;
    rtb_Product1_b4 = rtb_Product_m[3];
    if (rtb_Product_m[3] > rtb_Switch9_k) {
      rtb_Product1_b4 = rtb_Switch9_k;
    } else if (rtb_Product_m[3] < 0.0) {
      rtb_Product1_b4 = 0.0;
    }

    rtb_Product_m[3] = rtb_Product1_b4;
    Gen2_ref_DWork->u2_past[(int32_T)Gen2_ref_DWork->count - 1] = rtb_Product_m
      [1];
    Gen2_ref_DWork->count++;
    if (Gen2_ref_DWork->count > 100.0) {
      Gen2_ref_DWork->count = 1.0;
    }

    Gen2_ref_DWork->red_comp = true;
  }

  /* Sum: '<S749>/Sum' incorporates:
   *  Sum: '<S634>/Sum'
   */
  delta_y_tmp_tmp = rtb_Product_m[0] - rtb_Gain3;

  /* MATLAB Function: '<S749>/MATLAB Function' incorporates:
   *  Sum: '<S749>/Sum'
   */
  Gen2_ref_DWork->x_h -= 1.0 / Gen2_ref_B->BusInput3.SpeedCtrl.rTi_DPr_Limit *
    Gen2_ref_DWork->x_h * Gen2_ref_B->BusInput3.eng.Ts;
  if (delta_y_tmp_tmp > Gen2_ref_B->BusInput3.SpeedCtrl.rDPr_Limit) {
    Gen2_ref_DWork->SR_LoadStep = true;
    Gen2_ref_DWork->x_h = 1.0;
  } else if (delta_y_tmp_tmp < -Gen2_ref_B->BusInput3.SpeedCtrl.rDPr_Limit) {
    Gen2_ref_DWork->SR_LoadStep = false;
    Gen2_ref_DWork->x_h = 1.0;
  }

  rtb_Act = (Gen2_ref_DWork->x_h >
             Gen2_ref_B->BusInput3.SpeedCtrl.rDPr_Limit_Thrsh);

  /* Sum: '<S628>/Sum' incorporates:
   *  Sum: '<S634>/Sum1'
   *  Sum: '<S749>/Sum1'
   *  Sum: '<S8>/Sum'
   */
  rtb_Product1_c1_tmp = rtb_Switch_ks - rtb_Switch_i5[0];

  /* Switch: '<S628>/Switch' incorporates:
   *  Abs: '<S628>/Abs'
   *  Logic: '<S628>/Logical Operator'
   *  Logic: '<S628>/Logical Operator1'
   *  RelationalOperator: '<S628>/Relational Operator'
   *  Sum: '<S628>/Sum'
   */
  if ((!rtb_Act) && (Gen2_ref_B->BusInput3.SpeedCtrl.rN_thrshFiltLam > fabs
                     (rtb_Product1_c1_tmp))) {
    rtb_Product1_b4 = Gen2_ref_B->BusInput3.SpeedCtrl.rTi_LamCmd_iLQR;
  } else {
    rtb_Product1_b4 = Gen2_ref_B->BusInput3.eng.Ts;
  }

  /* End of Switch: '<S628>/Switch' */

  /* MATLAB Function: '<S628>/FILTER no delay' */
  Gen2_ref_FILTERnodelay(rtb_Product_m[1], rtb_Product1_b4,
    Gen2_ref_B->BusInput3.eng.Ts, rtb_bResetHlci,
    &Gen2_ref_B->sf_FILTERnodelay_b, &Gen2_ref_DWork->sf_FILTERnodelay_b, inst);

  /* Abs: '<S628>/Abs2' */
  rtb_Sum2_kg = fabs(Gen2_ref_B->BusInput3.SpeedCtrl.rNdbLambdaKp);

  /* Switch: '<S658>/Switch2' incorporates:
   *  Constant: '<S628>/  1'
   *  RelationalOperator: '<S658>/LowerRelop1'
   *  RelationalOperator: '<S658>/UpperRelop'
   *  Sum: '<S628>/Sum'
   *  Switch: '<S658>/Switch'
   */
  if (rtb_Product1_c1_tmp > 500.0) {
    rtb_Divide1_h4 = 500.0;
  } else if (rtb_Product1_c1_tmp < rtb_Sum2_kg) {
    /* Switch: '<S658>/Switch' */
    rtb_Divide1_h4 = rtb_Sum2_kg;
  } else {
    rtb_Divide1_h4 = rtb_Product1_c1_tmp;
  }

  /* End of Switch: '<S658>/Switch2' */

  /* Sum: '<S628>/Sum3' */
  rtb_Product1_fu = rtb_Divide1_h4 - rtb_Sum2_kg;

  /* Gain: '<S628>/Gain1' */
  rtb_Sum2_kg = rtb_Gain3;

  /* Switch: '<S659>/Switch' */
  if (Gen2_ref_B->BusInput3.SpeedCtrl.bGS_iLQR_addKpLam) {
    /* S-Function (sfix_look1_dyn): '<S659>/Lookup Table Dynamic2' */
    /* Dynamic Look-Up Table Block: '<S659>/Lookup Table Dynamic2'
     * Input0  Data Type:  Floating Point real_T
     * Input1  Data Type:  Floating Point real_T
     * Input2  Data Type:  Floating Point real_T
     * Output0 Data Type:  Floating Point real_T
     * Saturation Mode: Saturate
     * Lookup Method: Linear_Endpoint
     *
     */
    LookUp_real_T_real_T_SAT( &(rtb_LookupTableDynamic2_f),
      &Gen2_ref_B->BusInput3.SpeedCtrl.refPoint_addKpLam_Kp_y[0], rtb_Sum2_kg,
      &Gen2_ref_B->BusInput3.SpeedCtrl.refPoint_addKpLam_Kp_x[0], 5U, inst);
    rtb_Divide1_h4 = rtb_LookupTableDynamic2_f;
  } else {
    rtb_Divide1_h4 = Gen2_ref_B->BusInput3.SpeedCtrl.rGainLambdaKp;
  }

  /* End of Switch: '<S659>/Switch' */

  /* Product: '<S628>/Product1' incorporates:
   *  Abs: '<S628>/Abs1'
   *  Gain: '<S628>/Gain'
   */
  rtb_Product1_fu *= -0.001 * fabs(rtb_Divide1_h4);

  /* Switch: '<S659>/Switch1' */
  if (Gen2_ref_B->BusInput3.SpeedCtrl.bGS_iLQR_addKpLam) {
    /* S-Function (sfix_look1_dyn): '<S659>/Lookup Table Dynamic1' */
    /* Dynamic Look-Up Table Block: '<S659>/Lookup Table Dynamic1'
     * Input0  Data Type:  Floating Point real_T
     * Input1  Data Type:  Floating Point real_T
     * Input2  Data Type:  Floating Point real_T
     * Output0 Data Type:  Floating Point real_T
     * Saturation Mode: Saturate
     * Lookup Method: Linear_Endpoint
     *
     */
    LookUp_real_T_real_T_SAT( &(rtb_LookupTableDynamic1_h),
      &Gen2_ref_B->BusInput3.SpeedCtrl.refPoint_addKpLam_Ti_y[0], rtb_Sum2_kg,
      &Gen2_ref_B->BusInput3.SpeedCtrl.refPoint_addKpLam_Kp_x[0], 5U, inst);
    rtb_Sum2_kg = rtb_LookupTableDynamic1_h;
  } else {
    rtb_Sum2_kg = Gen2_ref_B->BusInput3.SpeedCtrl.rTiLambdaKp;
  }

  /* End of Switch: '<S659>/Switch1' */

  /* Outputs for Atomic SubSystem: '<S628>/Filter' */
  Gen2_ref_Filter3(rtb_Product1_fu, rtb_Sum2_kg, Gen2_ref_ConstB.Constant2,
                   rtb_bResetHlci, &Gen2_ref_B->Filter_b,
                   &Gen2_ref_DWork->Filter_b, inst);

  /* End of Outputs for SubSystem: '<S628>/Filter' */

  /* MinMax: '<S628>/MinMax' */
  if ((!(rtb_Product1_fu <= Gen2_ref_B->Filter_b.Switch)) && (!rtIsNaN
       (Gen2_ref_B->Filter_b.Switch))) {
    rtb_Product1_fu = Gen2_ref_B->Filter_b.Switch;
  }

  /* End of MinMax: '<S628>/MinMax' */

  /* Sum: '<S628>/Sum1' */
  rtb_Sum2_kg = Gen2_ref_B->sf_FILTERnodelay_b.y + rtb_Product1_fu;

  /* Switch: '<S657>/Switch2' incorporates:
   *  RelationalOperator: '<S657>/LowerRelop1'
   *  RelationalOperator: '<S657>/UpperRelop'
   *  Switch: '<S657>/Switch'
   */
  if (rtb_Sum2_kg > rtb_Switch2_n5) {
    rtb_Sum2_kg = rtb_Switch2_n5;
  } else if (rtb_Sum2_kg < rtb_Switch1_k) {
    /* Switch: '<S657>/Switch' */
    rtb_Sum2_kg = rtb_Switch1_k;
  }

  /* End of Switch: '<S657>/Switch2' */

  /* Switch: '<S8>/Switch12' incorporates:
   *  Constant: '<S8>/Constant4'
   *  Logic: '<S8>/Logical Operator6'
   *  Logic: '<S8>/Logical Operator8'
   */
  if ((!Gen2_ref_B->BusInput3.SpeedCtrl.bSwitchOutputSampleSS) ||
      Gen2_ref_B->TON2.LogicalOperator3) {
    Npred = Gen2_ref_B->BusInput3.SpeedCtrl.iOutputSample;
  } else {
    Npred = 1;
  }

  /* End of Switch: '<S8>/Switch12' */

  /* MATLAB Function: '<S8>/IntegerZOH' */
  Gen2_ref_IntegerZOH(rtb_Sum2_kg, Npred, &Gen2_ref_B->sf_IntegerZOH_g,
                      &Gen2_ref_DWork->sf_IntegerZOH_g, inst);

  /* Switch: '<Root>/lam_cmd' */
  if (rtb_LogicalOperator) {
    rtb_Product1_fu = Gen2_ref_B->sf_MATLABFunction1_h.LamOut;
  } else {
    rtb_Product1_fu = Gen2_ref_B->sf_IntegerZOH_g.y;
  }

  /* End of Switch: '<Root>/lam_cmd' */

  /* Outputs for Atomic SubSystem: '<S267>/lam2cg' */
  Gen2_ref_lam2cg1(rtb_Product1_fu, Gen2_ref_B->BusInput3.eng.rMin_Air_Ratio_kg,
                   &Gen2_ref_B->lam2cg, inst);

  /* End of Outputs for SubSystem: '<S267>/lam2cg' */

  /* Product: '<S267>/Divide3' incorporates:
   *  Bias: '<S267>/Bias'
   *  Constant: '<S267>/R_air'
   *  Product: '<S267>/Divide2'
   */
  rtb_Divide3_n_tmp = (Gen2_ref_B->Mg.Bias * Gen2_ref_B->lam2cg.Divide + 1.0) *
    287.15;

  /* Product: '<S267>/Divide' incorporates:
   *  Product: '<S267>/Divide3'
   *  Product: '<S268>/Divide'
   */
  rtb_SumofElements_l = rtb_Switch2_gd_idx_0 * Gen2_ref_B->BusInput3.eng.rVol_GM
    / Gen2_ref_B->T1LP_filt.Switch;
  R_2inp[0] = rtb_SumofElements_l / rtb_Divide3_n_tmp *
    Gen2_ref_B->BusInput3.fdc.rCF[0];
  rtb_RoundingFunction = rtb_Switch2_gd_idx_1 *
    Gen2_ref_B->BusInput3.eng.rVol_IC_LP / Gen2_ref_B->T1HP_filt.Switch;
  R_2inp[1] = rtb_RoundingFunction / rtb_Divide3_n_tmp *
    Gen2_ref_B->BusInput3.fdc.rCF[1];
  rtb_Switch2_d1 = rtb_Switch2_gd_idx_2 * Gen2_ref_B->BusInput3.eng.rVol_IC_HP /
    Gen2_ref_B->T2s_filt.Switch;
  R_2inp[2] = rtb_Switch2_d1 / rtb_Divide3_n_tmp * Gen2_ref_B->
    BusInput3.fdc.rCF[2];
  rtb_Product1_mqz = rtb_Switch2_gd_idx_3 * Gen2_ref_B->BusInput3.eng.rVol_im /
    Gen2_ref_B->T2s_filt.Switch;
  R_2inp[3] = rtb_Product1_mqz / rtb_Divide3_n_tmp *
    Gen2_ref_B->BusInput3.fdc.rCF[3];

  /* Product: '<S267>/Divide1' incorporates:
   *  Sum: '<S267>/Sum of Elements'
   */
  rtb_Divide1_h4 = (((R_2inp[0] + R_2inp[1]) + R_2inp[2]) + R_2inp[3]) *
    Gen2_ref_B->lam2cg.Divide;

  /* Switch: '<S267>/Switch' incorporates:
   *  Constant: '<S267>/Constant5'
   */
  if (Gen2_ref_B->BusInput3.fdc.bActive_dyn) {
    rtb_Switch2_l = rtb_Divide1_h4;
  } else {
    rtb_Switch2_l = 0.0;
  }

  /* End of Switch: '<S267>/Switch' */

  /* MATLAB Function: '<S305>/FILTER no delay4' */
  Gen2_ref_FILTERnodelay(rtb_DataTypeConversion15,
    Gen2_ref_B->BusInput3.fdc.rTiF_N_GF, Gen2_ref_B->BusInput3.eng.Ts,
    rtb_bResetBdc, &Gen2_ref_B->sf_FILTERnodelay4,
    &Gen2_ref_DWork->sf_FILTERnodelay4, inst);

  /* Outputs for Atomic SubSystem: '<S306>/2nd Order Filter4' */
  /* DiscreteIntegrator: '<S318>/Discrete-Time Integrator' */
  if (rtb_bResetBdc || (Gen2_ref_DWork->DiscreteTimeIntegrator_PrevR_i3 != 0)) {
    Gen2_ref_DWork->DiscreteTimeIntegrator_DSTAT_ic = 0.0;
  }

  rtb_SumofElements = Gen2_ref_DWork->DiscreteTimeIntegrator_DSTAT_ic;

  /* Product: '<S318>/Product' */
  rtb_Divide3_ep = Gen2_ref_B->BusInput3.fdc.r2ndOrdFiltOmegaSpeed *
    Gen2_ref_B->BusInput3.fdc.r2ndOrdFiltOmegaSpeed;

  /* Abs: '<S327>/Abs' */
  FILT_IN = fabs(rtb_Divide3_ep);

  /* Switch: '<S327>/Switch' incorporates:
   *  Constant: '<S327>/Constant2'
   *  RelationalOperator: '<S327>/Relational Operator'
   */
  if (2.2204460492503131E-16 >= FILT_IN) {
    delta_y = 2.2204460492503131E-16;
  } else {
    delta_y = rtb_Divide3_ep;
  }

  /* End of Switch: '<S327>/Switch' */

  /* Product: '<S318>/Divide1' */
  rtb_Sum4_g = rtb_DataTypeConversion15 / delta_y;

  /* DiscreteIntegrator: '<S318>/Discrete-Time Integrator1' */
  if (Gen2_ref_DWork->DiscreteTimeIntegrator1_IC_LO_n != 0) {
    Gen2_ref_DWork->DiscreteTimeIntegrator1_DSTAT_h = rtb_Sum4_g;
  }

  if (rtb_bResetBdc || (Gen2_ref_DWork->DiscreteTimeIntegrator1_Prev_ks != 0)) {
    Gen2_ref_DWork->DiscreteTimeIntegrator1_DSTAT_h = rtb_Sum4_g;
  }

  /* Product: '<S318>/Product1' incorporates:
   *  Constant: '<S318>/Constant1'
   */
  FILT_IN = Gen2_ref_B->BusInput3.fdc.r2ndOrdFiltOmegaSpeed *
    Gen2_ref_B->BusInput3.fdc.r2ndOrdFiltDSpeed * 2.0;

  /* Switch: '<S318>/Switch' incorporates:
   *  DiscreteIntegrator: '<S318>/Discrete-Time Integrator1'
   *  Product: '<S318>/Product2'
   *  RelationalOperator: '<S318>/Relational Operator'
   */
  if (rtb_Divide3_ep > 0.0) {
    rtb_Switch_kr = Gen2_ref_DWork->DiscreteTimeIntegrator1_DSTAT_h *
      rtb_Divide3_ep;
  } else {
    rtb_Switch_kr = rtb_DataTypeConversion15;
  }

  /* End of Switch: '<S318>/Switch' */

  /* Update for DiscreteIntegrator: '<S318>/Discrete-Time Integrator' incorporates:
   *  DiscreteIntegrator: '<S318>/Discrete-Time Integrator1'
   *  Product: '<S318>/Product3'
   *  Product: '<S318>/Product4'
   *  Sum: '<S318>/Sum'
   */
  Gen2_ref_DWork->DiscreteTimeIntegrator_DSTAT_ic += ((rtb_DataTypeConversion15
    - rtb_Divide3_ep * Gen2_ref_DWork->DiscreteTimeIntegrator1_DSTAT_h) -
    FILT_IN * Gen2_ref_DWork->DiscreteTimeIntegrator_DSTAT_ic) * 0.01;
  Gen2_ref_DWork->DiscreteTimeIntegrator_PrevR_i3 = (int8_T)rtb_bResetBdc;

  /* Update for DiscreteIntegrator: '<S318>/Discrete-Time Integrator1' incorporates:
   *  DiscreteIntegrator: '<S318>/Discrete-Time Integrator'
   */
  Gen2_ref_DWork->DiscreteTimeIntegrator1_IC_LO_n = 0U;
  Gen2_ref_DWork->DiscreteTimeIntegrator1_DSTAT_h += 0.01 * rtb_SumofElements;
  Gen2_ref_DWork->DiscreteTimeIntegrator1_Prev_ks = (int8_T)rtb_bResetBdc;

  /* End of Outputs for SubSystem: '<S306>/2nd Order Filter4' */

  /* Switch: '<S272>/Switch5' */
  if (Gen2_ref_B->BusInput3.fdc.bFiltdSpeedGasFlow) {
    /* Switch: '<S272>/Switch3' */
    if (Gen2_ref_B->BusInput3.fdc.bEnable2ndOrdFiltInputs) {
      /* Switch: '<S272>/Switch8' incorporates:
       *  Constant: '<S307>/Constant2'
       *  DiscreteIntegrator: '<S307>/Discrete-Time Integrator'
       *  Product: '<S307>/Product4'
       *  Product: '<S307>/Product5'
       *  Sum: '<S307>/Sum2'
       *  Sum: '<S307>/Sum4'
       */
      if (Gen2_ref_B->BusInput3.fdc.bEnableTransSwFilt) {
        rtb_Switch5_nn = (1.0 - Gen2_ref_DWork->DiscreteTimeIntegrator_DSTATE_d)
          * Gen2_ref_B->sf_FILTERnodelay4.y +
          Gen2_ref_DWork->DiscreteTimeIntegrator_DSTATE_d * rtb_Switch_kr;
      } else {
        rtb_Switch5_nn = rtb_Switch_kr;
      }

      /* End of Switch: '<S272>/Switch8' */
    } else {
      rtb_Switch5_nn = Gen2_ref_B->sf_FILTERnodelay4.y;
    }

    /* End of Switch: '<S272>/Switch3' */
  } else {
    rtb_Switch5_nn = rtb_DataTypeConversion15;
  }

  /* End of Switch: '<S272>/Switch5' */

  /* MATLAB Function: '<S305>/FILTER no delay5' */
  Gen2_ref_FILTERnodelay(rtb_p2s, Gen2_ref_B->BusInput3.fdc.rTiF_Pr_p2s_GF,
    Gen2_ref_B->BusInput3.eng.Ts, rtb_bResetBdc, &Gen2_ref_B->sf_FILTERnodelay5,
    &Gen2_ref_DWork->sf_FILTERnodelay5, inst);

  /* Switch: '<S272>/Switch4' */
  if (Gen2_ref_B->BusInput3.fdc.bFiltdPresGasFlow) {
    /* Switch: '<S272>/Switch1' */
    if (Gen2_ref_B->BusInput3.fdc.bEnable2ndOrdFiltInputs) {
      /* Switch: '<S272>/Switch7' incorporates:
       *  Constant: '<S307>/Constant2'
       *  DiscreteIntegrator: '<S307>/Discrete-Time Integrator'
       *  Product: '<S307>/Product2'
       *  Product: '<S307>/Product3'
       *  Sum: '<S307>/Sum1'
       *  Sum: '<S307>/Sum4'
       */
      if (Gen2_ref_B->BusInput3.fdc.bEnableTransSwFilt) {
        rtb_Switch4_p = (1.0 - Gen2_ref_DWork->DiscreteTimeIntegrator_DSTATE_d) *
          Gen2_ref_B->sf_FILTERnodelay5.y +
          Gen2_ref_DWork->DiscreteTimeIntegrator_DSTATE_d *
          Gen2_ref_B->undOrderFilter3.Switch;
      } else {
        rtb_Switch4_p = Gen2_ref_B->undOrderFilter3.Switch;
      }

      /* End of Switch: '<S272>/Switch7' */
    } else {
      rtb_Switch4_p = Gen2_ref_B->sf_FILTERnodelay5.y;
    }

    /* End of Switch: '<S272>/Switch1' */
  } else {
    rtb_Switch4_p = rtb_p2s;
  }

  /* End of Switch: '<S272>/Switch4' */

  /* Outputs for Atomic SubSystem: '<S267>/lam2cg1' */
  Gen2_ref_lam2cg1_a(rtb_Product1_fu, Gen2_ref_B->BusInput3.eng.rMin_Air_Ratio,
                     &Gen2_ref_B->lam2cg1_a, inst);

  /* End of Outputs for SubSystem: '<S267>/lam2cg1' */

  /* Switch: '<S273>/Switch' incorporates:
   *  Constant: '<S273>/Constant2'
   *  RelationalOperator: '<S273>/Relational Operator'
   */
  if (1.0 >= rtb_bResetHlci_0) {
    delta_y = 1.0;
  } else {
    delta_y = Gen2_ref_B->T2s_filt.Switch;
  }

  /* End of Switch: '<S273>/Switch' */

  /* Gain: '<S267>/Gain2' incorporates:
   *  Gain: '<S144>/Gain2'
   *  Gain: '<S268>/Gain2'
   */
  rtb_Gain_kp = 0.5 * Gen2_ref_B->BusInput3.eng.rVol_Hub_Eng;

  /* Product: '<S267>/Divide8' incorporates:
   *  Gain: '<S267>/Gain1'
   *  Product: '<S268>/Divide8'
   */
  rtb_Sum_e = 0.016666666666666666 * rtb_Switch5_nn * rtb_etaVolConst_lt;

  /* Product: '<S267>/Product3' incorporates:
   *  Gain: '<S267>/Gain2'
   *  Gain: '<S267>/StandardCond'
   *  Product: '<S267>/Divide10'
   *  Product: '<S267>/Divide8'
   */
  rtb_Product3_g = rtb_Switch4_p / delta_y * 0.0026957809030347889 * rtb_Sum_e *
    Gen2_ref_B->lam2cg1_a.Divide * rtb_Gain_kp *
    Gen2_ref_B->BusInput3.eng.rRho_gas;

  /* Sum: '<S267>/Add1' */
  rtb_SumofElements = rtb_Switch2_l + rtb_Product3_g;

  /* Sum: '<S5>/Add' incorporates:
   *  Constant: '<S11>/Constant'
   *  Sum: '<S11>/Sum'
   */
  rtb_Switch2_l = 1.0 - Gen2_ref_B->BusInput.IN_EC_rGT_RatioMix_TC2;

  /* Switch: '<S5>/Switch12' incorporates:
   *  Constant: '<S5>/Constant4'
   *  Logic: '<S5>/Logical Operator6'
   *  Logic: '<S5>/Logical Operator8'
   */
  if ((!Gen2_ref_B->BusInput3.fdc.bSwitchOutputSampleSS) ||
      Gen2_ref_B->TON2.LogicalOperator3) {
    Npred = Gen2_ref_B->BusInput3.fdc.iOutputSample;
  } else {
    Npred = 1;
  }

  /* End of Switch: '<S5>/Switch12' */

  /* MATLAB Function: '<S5>/IntegerZOH' incorporates:
   *  Product: '<S5>/Divide'
   */
  Gen2_ref_IntegerZOH(rtb_SumofElements * rtb_Switch2_l, Npred,
                      &Gen2_ref_B->sf_IntegerZOH_f,
                      &Gen2_ref_DWork->sf_IntegerZOH_f, inst);

  /* Product: '<S494>/delta rise limit' incorporates:
   *  SampleTimeMath: '<S494>/sample time'
   *
   * About '<S494>/sample time':
   *  y = K where K = ( w * Ts )
   */
  rtb_Switch2_l = Gen2_ref_B->BusInput3.LR.rRL_GasFlowSatCompUp * 0.01;

  /* UnitDelay: '<Root>/Unit Delay4' */
  rtb_Divide3_ep = Gen2_ref_DWork->UnitDelay4_DSTATE;

  /* Switch: '<S1>/Switch8' */
  if (Gen2_ref_B->BusInput3.bdcMisc.bUnfilteredFeedback) {
    rtb_MassFlowCalc = rtb_p2s;
  } else {
    rtb_MassFlowCalc = Gen2_ref_B->p2s_filt.Switch;
  }

  /* End of Switch: '<S1>/Switch8' */

  /* Outputs for Atomic SubSystem: '<S204>/p2HP_filt' */
  Gen2_ref_N_TC_HP_filt(rtb_p2HP, Gen2_ref_B->BusInput3.inFilt.rTiF_Pr,
                        rtb_bResetBdc, &Gen2_ref_B->p2HP_filt,
                        &Gen2_ref_DWork->p2HP_filt, inst);

  /* End of Outputs for SubSystem: '<S204>/p2HP_filt' */

  /* Switch: '<S1>/Switch9' */
  if (Gen2_ref_B->BusInput3.bdcMisc.bUnfilteredFeedback) {
    rtb_Switch2_a = rtb_p2HP;
  } else {
    rtb_Switch2_a = Gen2_ref_B->p2HP_filt.Switch;
  }

  /* End of Switch: '<S1>/Switch9' */

  /* Switch: '<S32>/Switch' incorporates:
   *  Abs: '<S32>/Abs'
   *  Constant: '<S32>/Constant2'
   *  RelationalOperator: '<S32>/Relational Operator'
   */
  if (0.1 >= fabs(rtb_Switch2_a)) {
    delta_y = 0.1;
  } else {
    delta_y = rtb_Switch2_a;
  }

  /* End of Switch: '<S32>/Switch' */

  /* Product: '<S1>/Divide' */
  rtb_Divide_br = rtb_MassFlowCalc / delta_y;

  /* Outputs for Atomic SubSystem: '<S202>/p1HP_filt' */
  Gen2_ref_N_TC_HP_filt(rtb_p1HP, Gen2_ref_B->BusInput3.inFilt.rTiF_Pr,
                        rtb_bResetBdc, &Gen2_ref_B->p1HP_filt,
                        &Gen2_ref_DWork->p1HP_filt, inst);

  /* End of Outputs for SubSystem: '<S202>/p1HP_filt' */

  /* Switch: '<S1>/Switch10' incorporates:
   *  Constant: '<S1>/Constant2'
   *  Switch: '<S1>/Switch11'
   */
  if (Gen2_ref_B->BusInput3.bdcMisc.bUnfilteredFeedback) {
    rtb_Switch2_oou = rtb_p1HP;
    x = rtb_p1LP;
  } else {
    rtb_Switch2_oou = Gen2_ref_B->p1HP_filt.Switch;
    x = 100000.0;
  }

  /* End of Switch: '<S1>/Switch10' */

  /* Abs: '<S34>/Abs' incorporates:
   *  Abs: '<S35>/Abs'
   */
  rtb_p1LP = fabs(x);
  rtb_Switch_n = rtb_p1LP;

  /* Switch: '<S34>/Switch' incorporates:
   *  Constant: '<S34>/Constant2'
   *  RelationalOperator: '<S34>/Relational Operator'
   */
  if (0.1 >= rtb_Switch_n) {
    delta_y = 0.1;
  } else {
    delta_y = x;
  }

  /* End of Switch: '<S34>/Switch' */

  /* Product: '<S1>/Divide2' */
  rtb_Divide2 = rtb_Switch2_oou / delta_y;

  /* Abs: '<S33>/Abs' */
  rtb_Switch_n = fabs(rtb_Switch2_oou);

  /* Switch: '<S33>/Switch' incorporates:
   *  Constant: '<S33>/Constant2'
   *  RelationalOperator: '<S33>/Relational Operator'
   */
  if (0.1 >= rtb_Switch_n) {
    rtb_Switch2_oou = 0.1;
  }

  /* End of Switch: '<S33>/Switch' */

  /* Product: '<S1>/Divide1' */
  rtb_Divide1_fn = rtb_Switch2_a / rtb_Switch2_oou;

  /* Abs: '<S35>/Abs' */
  rtb_Switch_n = rtb_p1LP;

  /* Switch: '<S35>/Switch' incorporates:
   *  Constant: '<S35>/Constant2'
   *  RelationalOperator: '<S35>/Relational Operator'
   */
  if (0.1 >= rtb_Switch_n) {
    x = 0.1;
  }

  /* End of Switch: '<S35>/Switch' */

  /* Product: '<S1>/Divide3' */
  rtb_Divide3_a0 = rtb_MassFlowCalc / x;

  /* MATLAB Function: '<S24>/MATLAB Function' incorporates:
   *  Gain: '<S24>/Gain'
   *  Sum: '<S24>/Sum'
   */
  Gen2_ref_MATLABFunction(1.0E-5 * Gen2_ref_B->p2s_filt.Switch,
    Gen2_ref_B->BusInput3.bdcMisc.rPrSwitchFFmethod,
    Gen2_ref_B->BusInput3.bdcMisc.rPrSwitchFFmethod +
    Gen2_ref_B->BusInput3.bdcMisc.rPrSwitchFFmethod_hys,
    &Gen2_ref_B->sf_MATLABFunction_f, &Gen2_ref_DWork->sf_MATLABFunction_f, inst);

  /* Abs: '<S139>/Abs' */
  rtb_Switch_n = fabs(Gen2_ref_B->BusInput3.eng.rNum_TCperStage);

  /* Switch: '<S139>/Switch' incorporates:
   *  Constant: '<S139>/Constant2'
   *  RelationalOperator: '<S139>/Relational Operator'
   */
  if (2.2204460492503131E-16 >= rtb_Switch_n) {
    rtb_Switch_n = 2.2204460492503131E-16;
  } else {
    rtb_Switch_n = Gen2_ref_B->BusInput3.eng.rNum_TCperStage;
  }

  /* End of Switch: '<S139>/Switch' */

  /* Gain: '<S144>/Gain1' */
  x = 0.016666666666666666 * rtb_DataTypeConversion15;

  /* Outputs for Atomic SubSystem: '<S144>/lam2cg1' */
  Gen2_ref_lam2cg1(rtb_Product1_fu, Gen2_ref_B->BusInput3.eng.rMin_Air_Ratio,
                   &Gen2_ref_B->lam2cg1, inst);

  /* End of Outputs for SubSystem: '<S144>/lam2cg1' */

  /* Gain: '<S144>/Gain2' */
  rtb_Switch2_a = rtb_Gain_kp;

  /* Switch: '<S149>/Switch' incorporates:
   *  Constant: '<S149>/Constant2'
   *  RelationalOperator: '<S149>/Relational Operator'
   */
  if (2.2204460492503131E-16 >= rtb_bResetHlci_0) {
    delta_y = 2.2204460492503131E-16;
  } else {
    delta_y = Gen2_ref_B->T2s_filt.Switch;
  }

  /* End of Switch: '<S149>/Switch' */

  /* Fcn: '<S144>/MassFlowCalc' incorporates:
   *  Constant: '<S144>/rhoAir'
   *  Gain: '<S144>/StandardCond'
   *  Product: '<S144>/Divide10'
   */
  rtb_MassFlowCalc = Gen2_ref_B->p2s_filt.Switch / delta_y *
    0.0026957809030347889 * (rtb_etaVolConst_lt * x) * rtb_Switch2_a * ((1.0 -
    Gen2_ref_B->lam2cg1.Divide) * 1.293 + Gen2_ref_B->lam2cg1.Divide *
    Gen2_ref_B->BusInput3.eng.rRho_gas);

  /* Logic: '<S1>/Logical Operator1' */
  rtb_LogicalOperator_hi = (Gen2_ref_B->BusInput3.bdcMisc.bReset_Filter ||
    Gen2_ref_B->BusInput3.bdcMisc.bActive_BDC);

  /* Sum: '<S31>/Diff' incorporates:
   *  UnitDelay: '<S31>/UD'
   */
  u0_0 = (uint8_T)(rtb_LogicalOperator_hi - Gen2_ref_DWork->UD_DSTATE);

  /* Saturate: '<S1>/Saturation1' */
  if (u0_0 > 1) {
    u0_0 = 1U;
  }

  /* End of Saturate: '<S1>/Saturation1' */

  /* Logic: '<S1>/Logical Operator2' incorporates:
   *  DataTypeConversion: '<S1>/Data Type Conversion21'
   */
  rtb_LogicalOperator2_dc = (rtb_bResetBdc || (u0_0 != 0));

  /* Outputs for Atomic SubSystem: '<S134>/Filter' */
  /* UnitDelay: '<S1>/Unit Delay1' */
  Gen2_ref_Filter3(Gen2_ref_DWork->UnitDelay1_DSTATE_ek,
                   Gen2_ref_B->BusInput3.SpeedCtrl.rTi_CBV_SurgeProtec,
                   Gen2_ref_ConstB.u, rtb_LogicalOperator2_dc,
                   &Gen2_ref_B->Filter, &Gen2_ref_DWork->Filter, inst);

  /* End of Outputs for SubSystem: '<S134>/Filter' */

  /* Lookup_n-D: '<S134>/LT%2deg' incorporates:
   *  Switch: '<S141>/Switch'
   */
  x = look1_binlxpw(Gen2_ref_B->Filter.Switch, Gen2_ref_ConstP.LT2deg_bp01Data,
                    Gen2_ref_ConstP.LT2deg_tableData, 3U, inst);

  /* S-Function (sfix_look1_dyn): '<S134>/Lookup Table Dynamic' */
  /* Dynamic Look-Up Table Block: '<S134>/Lookup Table Dynamic'
   * Input0  Data Type:  Floating Point real_T
   * Input1  Data Type:  Floating Point real_T
   * Input2  Data Type:  Floating Point real_T
   * Output0 Data Type:  Floating Point real_T
   * Lookup Method: Linear_Endpoint
   *
   */
  LookUp_real_T_real_T( &(rtb_LookupTableDynamic),
                       &Gen2_ref_B->BusInput3.bdcCbv.rCd_vect_y[0], x,
                       &Gen2_ref_B->BusInput3.bdcCbv.rCd_vect_x[0], 10U, inst);

  /* MATLAB Function: '<S134>/MATLAB Function1' incorporates:
   *  Constant: '<S134>/Constant3'
   *  Constant: '<S1>/Constant2'
   *  Product: '<S134>/Product1'
   */
  if (Gen2_ref_B->p2HP_filt.Switch >= 100000.0) {
    if ((1.0E-6 >= Gen2_ref_B->p2HP_filt.Switch) || rtIsNaN
        (Gen2_ref_B->p2HP_filt.Switch)) {
      delta_y = 1.0E-6;
    } else {
      delta_y = Gen2_ref_B->p2HP_filt.Switch;
    }

    r = 100000.0 / delta_y;
    if ((1.0E-6 >= r) || rtIsNaN(r)) {
      r = 1.0E-6;
    }

    if (1.0 / r <= 1.8929291587378541) {
      u1 = sqrt(287.15 * Gen2_ref_B->T2s_filt.Switch);
      if ((1.0E-6 >= u1) || rtIsNaN(u1)) {
        u1 = 1.0E-6;
      }

      rtb_p1LP = 0.78539816339744828 * Gen2_ref_B->BusInput3.bdcCbv.rDref *
        Gen2_ref_B->BusInput3.bdcCbv.rDref * rtb_LookupTableDynamic *
        Gen2_ref_B->p2HP_filt.Switch / u1 * sqrt((rt_powd_snf(r,
        1.4285714285714286, inst) - rt_powd_snf(r, 1.7142857142857144, inst)) *
        7.0000000000000009);
    } else {
      u1 = sqrt(287.15 * Gen2_ref_B->T2s_filt.Switch);
      if ((1.0E-6 >= u1) || rtIsNaN(u1)) {
        u1 = 1.0E-6;
      }

      rtb_p1LP = 0.78539816339744828 * Gen2_ref_B->BusInput3.bdcCbv.rDref *
        Gen2_ref_B->BusInput3.bdcCbv.rDref * rtb_LookupTableDynamic *
        Gen2_ref_B->p2HP_filt.Switch / u1 * 0.6847314563772704;
    }
  } else {
    rtb_p1LP = 0.0;
  }

  /* End of MATLAB Function: '<S134>/MATLAB Function1' */

  /* Product: '<S134>/Divide1' */
  x = rtb_p1LP * Gen2_ref_B->BusInput3.eng.rNum_CBV;

  /* Fcn: '<S134>/CorredtedMassflow' incorporates:
   *  Product: '<S134>/Divide'
   *  Sum: '<S134>/Add2'
   *  UnitDelay: '<Root>/Unit Delay2'
   */
  rtb_p1LP = Gen2_ref_B->T1LP_filt.Switch / 298.0;
  if (rtb_p1LP < 0.0) {
    rtb_p1LP = -sqrt(-rtb_p1LP);
  } else {
    rtb_p1LP = sqrt(rtb_p1LP);
  }

  rtb_Switch_n = (((rtb_MassFlowCalc + x) + Gen2_ref_DWork->UnitDelay2_DSTATE_h
                   [2]) + Gen2_ref_DWork->UnitDelay2_DSTATE_h[3]) * (1.0 /
    rtb_Switch_n) * rtb_p1LP * 100000.0 / 100000.0;

  /* End of Fcn: '<S134>/CorredtedMassflow' */

  /* Fcn: '<S134>/SurgeLine1' */
  rtb_Saturation_gh = Gen2_ref_B->BusInput3.SpeedCtrl.rK_SurgeLine_LP *
    rtb_Switch_n + Gen2_ref_B->BusInput3.SpeedCtrl.rA_SurgeLine_LP;

  /* Saturate: '<S134>/Saturation' */
  if (rtb_Saturation_gh > 7.0) {
    rtb_Saturation_gh = 7.0;
  } else if (rtb_Saturation_gh < 1.0) {
    rtb_Saturation_gh = 1.0;
  }

  /* End of Saturate: '<S134>/Saturation' */

  /* Switch: '<S1>/Switch7' */
  if (Gen2_ref_B->BusInput3.SpeedCtrl.bSwitch_SurgeLine_LIMIT) {
    /* Switch: '<S43>/Switch1' */
    if (Gen2_ref_B->BusInput3.SpeedCtrl.bSwitch_SurgeLine_LIMIT) {
      rtb_p1LP = rtb_Saturation_gh;
    } else {
      rtb_p1LP = Gen2_ref_B->BusInput3.traj.rPr_p2s_max;
    }

    /* End of Switch: '<S43>/Switch1' */
  } else {
    rtb_p1LP = Gen2_ref_B->BusInput3.traj.rPr_p2s_max;
  }

  /* End of Switch: '<S1>/Switch7' */

  /* Switch: '<S58>/Switch2' incorporates:
   *  RelationalOperator: '<S58>/LowerRelop1'
   *  RelationalOperator: '<S58>/UpperRelop'
   *  Switch: '<S58>/Switch'
   */
  if (rtb_p1LP > Gen2_ref_B->BusInput3.traj.rPr_p2s_max) {
    rtb_Switch2_oou = Gen2_ref_B->BusInput3.traj.rPr_p2s_max;
  } else if (rtb_p1LP < Gen2_ref_B->BusInput3.bdcMisc.rMinLimSurgeline) {
    /* Switch: '<S58>/Switch' */
    rtb_Switch2_oou = Gen2_ref_B->BusInput3.bdcMisc.rMinLimSurgeline;
  } else {
    rtb_Switch2_oou = rtb_p1LP;
  }

  /* End of Switch: '<S58>/Switch2' */

  /* UnitDelay: '<S62>/Unit Delay4' */
  rtb_LogicalOperator2_ov = Gen2_ref_DWork->UnitDelay4_DSTATE_k;

  /* Gain: '<S23>/Gain' */
  rtb_Gain_kl = rtb_kW2W1_h;
  for (i = 0; i < 5; i++) {
    /* Sum: '<S23>/Sum12' incorporates:
     *  Sum: '<S23>/Sum8'
     *  Sum: '<S25>/Sum2'
     *  Switch: '<S106>/Switch2'
     */
    rtb_Gain1_eu[i] = Gen2_ref_B->BusInput3.traj.rOffs_WS_Actuators +
      Gen2_ref_B->BusInput3.traj.rPrR_deltaP_TV_x[i];
  }

  /* S-Function (sfix_look1_dyn): '<S23>/Lookup Table Dynamic' */
  /* Dynamic Look-Up Table Block: '<S23>/Lookup Table Dynamic'
   * Input0  Data Type:  Floating Point real_T
   * Input1  Data Type:  Floating Point real_T
   * Input2  Data Type:  Floating Point real_T
   * Output0 Data Type:  Floating Point real_T
   * Lookup Method: Linear_Endpoint
   *
   */
  LookUp_real_T_real_T( &(rtb_Switch2_a),
                       &Gen2_ref_B->BusInput3.traj.rPrR_deltaP_TV_y[0],
                       rtb_Gain_kl, &rtb_Gain1_eu[0], 4U, inst);

  /* Saturate: '<S23>/Saturation1' */
  if (Gen2_ref_B->BusInput3.eng.rNum_TV > 1.0) {
    /* Saturate: '<S44>/Saturation' incorporates:
     *  Saturate: '<S25>/Saturation1'
     *  Switch: '<S106>/Switch2'
     */
    rtb_Saturation1_i = 1.0;
  } else if (Gen2_ref_B->BusInput3.eng.rNum_TV < 0.0) {
    /* Saturate: '<S44>/Saturation' incorporates:
     *  Saturate: '<S25>/Saturation1'
     *  Switch: '<S106>/Switch2'
     */
    rtb_Saturation1_i = 0.0;
  } else {
    /* Saturate: '<S44>/Saturation' incorporates:
     *  Saturate: '<S25>/Saturation1'
     *  Switch: '<S106>/Switch2'
     */
    rtb_Saturation1_i = Gen2_ref_B->BusInput3.eng.rNum_TV;
  }

  rtb_MinMax_a = rtb_Saturation1_i;

  /* End of Saturate: '<S23>/Saturation1' */

  /* Product: '<S23>/Product2' */
  rtb_Product2 = rtb_Switch2_a * rtb_MinMax_a;

  /* MATLAB Function: '<S62>/MATLAB Function' */
  Gen2_ref_DWork->x_i = ((rtb_Product2 < Gen2_ref_B->BusInput3.traj.rDPp2sCompON)
    || ((!(rtb_Product2 > Gen2_ref_B->BusInput3.traj.rDPp2sCompON + 0.03)) &&
        Gen2_ref_DWork->x_i));

  /* Logic: '<S62>/Logical Operator' incorporates:
   *  Logic: '<S62>/Logical Operator9'
   *  MATLAB Function: '<S62>/MATLAB Function'
   */
  rtb_LogicalOperator_aw = ((!rtb_LogicalOperator2_ov) || (!Gen2_ref_DWork->x_i));

  /* Logic: '<S62>/Logical Operator1' incorporates:
   *  Logic: '<S62>/Logical Operator2'
   */
  rtb_LogicalOperator1_i2 = ((rtb_LogicalOperator_aw &&
    Gen2_ref_B->BusInput3.traj.bResetCompTrans) || rtb_LogicalOperator2_dc);

  /* DiscreteIntegrator: '<S62>/Discrete-Time Integrator' */
  if (rtb_LogicalOperator1_i2 ||
      (Gen2_ref_DWork->DiscreteTimeIntegrator_PrevR_oa != 0)) {
    Gen2_ref_DWork->DiscreteTimeIntegrator_DSTATE_a = 0.0;
  }

  if (Gen2_ref_DWork->DiscreteTimeIntegrator_DSTATE_a >= 1.0) {
    Gen2_ref_DWork->DiscreteTimeIntegrator_DSTATE_a = 1.0;
  } else if (Gen2_ref_DWork->DiscreteTimeIntegrator_DSTATE_a <= -0.1) {
    Gen2_ref_DWork->DiscreteTimeIntegrator_DSTATE_a = -0.1;
  }

  /* Product: '<S88>/delta rise limit' incorporates:
   *  Constant: '<S78>/Constant1'
   *  SampleTimeMath: '<S88>/sample time'
   *
   * About '<S88>/sample time':
   *  y = K where K = ( w * Ts )
   */
  rtb_MinMax_a = 1.0E+8;

  /* Switch: '<Root>/BDC_traj' incorporates:
   *  Gain: '<S431>/Gain4'
   */
  if (!rtb_LogicalOperator) {
    rtb_Pa2bar_o = 100000.0 * rtb_Product_m[0];
  }

  /* End of Switch: '<Root>/BDC_traj' */

  /* Gain: '<S23>/Gain1' */
  rtb_p1LP = 1.0E-5 * rtb_Pa2bar_o;

  /* Logic: '<S78>/Logical Operator' incorporates:
   *  RelationalOperator: '<S78>/Relational Operator'
   */
  rtb_LogicalOperator2_p1 = (Gen2_ref_B->BusInput3.traj.bRateLimRejON &&
    (Gen2_ref_B->BusInput3.traj.rNmaxRateLimRejON > rtb_DataTypeConversion15));

  /* Logic: '<S78>/Logical Operator1' incorporates:
   *  Logic: '<S78>/Logical Operator2'
   */
  rtb_LogicalOperator1_a0 = ((!rtb_LogicalOperator2_p1) ||
    rtb_LogicalOperator2_dc);

  /* Gain: '<S23>/Gain2' */
  rtb_p1HP = 1.0E-5 * rtb_Divide_kt;

  /* Gain: '<S78>/Gain' */
  rtb_Divide_kt = 100.0 * Gen2_ref_B->BusInput3.traj.rTi_RateLimRej;

  /* Delay: '<S78>/Variable Integer Delay' */
  Gen2_ref_DWork->icLoad_ev =
    ((((Gen2_ref_PrevZCSigState->VariableIntegerDelay_Reset_ZC_i == 1) !=
       (int32_T)rtb_LogicalOperator1_a0) &&
      (Gen2_ref_PrevZCSigState->VariableIntegerDelay_Reset_ZC_i != 3)) ||
     rtb_LogicalOperator1_a0 || Gen2_ref_DWork->icLoad_ev);
  Gen2_ref_PrevZCSigState->VariableIntegerDelay_Reset_ZC_i =
    rtb_LogicalOperator1_a0;
  if (Gen2_ref_DWork->icLoad_ev) {
    for (i = 0; i < 300; i++) {
      Gen2_ref_DWork->VariableIntegerDelay_DSTATE_b[i] = rtb_p1HP;
    }
  }

  if ((rtb_Divide_kt < 1.0) || rtIsNaN(rtb_Divide_kt)) {
    rtb_VariableIntegerDelay_b = rtb_p1HP;
  } else {
    if (rtb_Divide_kt > 300.0) {
      i = 300;
    } else {
      delta_y = floor(rtb_Divide_kt);
      if (rtIsNaN(delta_y)) {
        i = 0;
      } else {
        i = (int32_T)(uint32_T)fmod(delta_y, 4.294967296E+9);
      }
    }

    rtb_VariableIntegerDelay_b = Gen2_ref_DWork->VariableIntegerDelay_DSTATE_b
      [300U - i];
  }

  /* Saturate: '<S78>/Saturation' */
  if (Gen2_ref_B->BusInput3.traj.rTi_RateLimRej <= 0.01) {
    rtb_Switch2_a = 0.01;
  } else {
    rtb_Switch2_a = Gen2_ref_B->BusInput3.traj.rTi_RateLimRej;
  }

  /* End of Saturate: '<S78>/Saturation' */

  /* Product: '<S78>/Divide' incorporates:
   *  Sum: '<S78>/Sum'
   */
  rtb_Divide_kt = (rtb_p1HP - rtb_VariableIntegerDelay_b) / rtb_Switch2_a;

  /* Abs: '<S78>/Abs2' incorporates:
   *  Abs: '<S77>/Abs2'
   */
  rtb_UkYk1_a4 = fabs(Gen2_ref_B->BusInput3.traj.rPrTriggerRateLimRej);

  /* Gain: '<S78>/Gain3' incorporates:
   *  Abs: '<S78>/Abs2'
   */
  rtb_Switch2_jq = -rtb_UkYk1_a4;

  /* Logic: '<S78>/Logical Operator3' incorporates:
   *  RelationalOperator: '<S78>/Relational Operator1'
   */
  rtb_LogicalOperator3_ja = (rtb_LogicalOperator1_a0 || (rtb_Divide_kt >
    rtb_Switch2_jq));

  /* Delay: '<S88>/Delay' */
  Gen2_ref_DWork->icLoad_d = ((((Gen2_ref_PrevZCSigState->Delay_Reset_ZCE_d == 1)
    != (int32_T)rtb_LogicalOperator3_ja) &&
    (Gen2_ref_PrevZCSigState->Delay_Reset_ZCE_d != 3)) ||
    rtb_LogicalOperator3_ja || Gen2_ref_DWork->icLoad_d);
  Gen2_ref_PrevZCSigState->Delay_Reset_ZCE_d = rtb_LogicalOperator3_ja;
  if (Gen2_ref_DWork->icLoad_d) {
    Gen2_ref_DWork->Delay_DSTATE_ko = rtb_p1LP;
  }

  /* Switch: '<S88>/etaVolConst' incorporates:
   *  UnitDelay: '<S78>/Unit Delay'
   */
  if (rtb_LogicalOperator3_ja) {
    rtb_p2HP = rtb_p1LP;
  } else {
    rtb_p2HP = Gen2_ref_DWork->UnitDelay_DSTATE_e;
  }

  /* End of Switch: '<S88>/etaVolConst' */

  /* Sum: '<S88>/Difference Inputs1' incorporates:
   *  Delay: '<S88>/Delay'
   */
  rtb_p2HP -= Gen2_ref_DWork->Delay_DSTATE_ko;

  /* Abs: '<S78>/Abs1' */
  rtb_Sum1_dh = fabs(Gen2_ref_B->BusInput3.traj.rPrDeltaMinRateLimRej);

  /* Abs: '<S78>/Abs' incorporates:
   *  Abs: '<S77>/Abs'
   */
  rtb_Switch_czo = fabs(Gen2_ref_B->BusInput3.traj.rPrDeltaMinRateLimRejFF);

  /* Product: '<S78>/Divide1' incorporates:
   *  Abs: '<S78>/Abs'
   *  Gain: '<S78>/Gain1'
   */
  rtb_MinMax_mf = -rtb_Switch_czo / rtb_Switch2_a;

  /* MinMax: '<S78>/MinMax' */
  if ((rtb_Divide_kt <= rtb_MinMax_mf) || rtIsNaN(rtb_MinMax_mf)) {
    rtb_MinMax_mf = rtb_Divide_kt;
  }

  /* End of MinMax: '<S78>/MinMax' */

  /* Product: '<S78>/Divide2' incorporates:
   *  Gain: '<S78>/Gain2'
   */
  rtb_MinMax3 = -rtb_Sum1_dh / rtb_Switch2_a;

  /* MinMax: '<S78>/MinMax3' */
  if ((!(rtb_MinMax3 <= rtb_MinMax_mf)) && (!rtIsNaN(rtb_MinMax_mf))) {
    rtb_MinMax3 = rtb_MinMax_mf;
  }

  /* End of MinMax: '<S78>/MinMax3' */

  /* Switch: '<S92>/Switch2' incorporates:
   *  RelationalOperator: '<S92>/LowerRelop1'
   */
  if (!(rtb_p2HP > 1.0E+8)) {
    /* Product: '<S88>/delta fall limit' incorporates:
     *  SampleTimeMath: '<S88>/sample time'
     *
     * About '<S88>/sample time':
     *  y = K where K = ( w * Ts )
     */
    rtb_Sum4_g = rtb_MinMax3 * 0.01;

    /* Switch: '<S92>/Switch' incorporates:
     *  RelationalOperator: '<S92>/UpperRelop'
     */
    if (rtb_p2HP < rtb_Sum4_g) {
      rtb_MinMax_a = rtb_Sum4_g;
    } else {
      rtb_MinMax_a = rtb_p2HP;
    }

    /* End of Switch: '<S92>/Switch' */
  }

  /* End of Switch: '<S92>/Switch2' */

  /* Sum: '<S88>/Difference Inputs2' incorporates:
   *  Delay: '<S88>/Delay'
   */
  rtb_p2HP = rtb_MinMax_a + Gen2_ref_DWork->Delay_DSTATE_ko;

  /* Product: '<S90>/delta rise limit' incorporates:
   *  Constant: '<S78>/Constant4'
   *  SampleTimeMath: '<S90>/sample time'
   *
   * About '<S90>/sample time':
   *  y = K where K = ( w * Ts )
   */
  rtb_Sum_c = 1.0E+8;

  /* Delay: '<S90>/Delay' incorporates:
   *  Delay: '<S78>/Variable Integer Delay'
   */
  Gen2_ref_DWork->icLoad_es = ((((Gen2_ref_PrevZCSigState->Delay_Reset_ZCE_l ==
    1) != (int32_T)rtb_LogicalOperator1_a0) &&
    (Gen2_ref_PrevZCSigState->Delay_Reset_ZCE_l != 3)) ||
    rtb_LogicalOperator1_a0 || Gen2_ref_DWork->icLoad_es);
  Gen2_ref_PrevZCSigState->Delay_Reset_ZCE_l = rtb_LogicalOperator1_a0;
  if (Gen2_ref_DWork->icLoad_es) {
    Gen2_ref_DWork->Delay_DSTATE_j = rtb_p1LP;
  }

  /* Sum: '<S90>/Difference Inputs1' incorporates:
   *  Delay: '<S90>/Delay'
   *  Switch: '<S90>/etaVolConst'
   */
  rtb_Sum4_g = rtb_p1LP - Gen2_ref_DWork->Delay_DSTATE_j;

  /* Gain: '<S78>/Gain5' incorporates:
   *  Gain: '<S77>/Gain5'
   */
  FILT_IN = 0.001 * Gen2_ref_B->BusInput3.leanox.rPr_mbar_2;
  rtb_Sum1_dh = FILT_IN;

  /* Gain: '<S78>/Gain6' incorporates:
   *  Product: '<S78>/Divide3'
   */
  rtb_Switch9_k = -(rtb_Sum1_dh / rtb_Switch2_a);

  /* Switch: '<S94>/Switch2' incorporates:
   *  RelationalOperator: '<S94>/LowerRelop1'
   */
  if (!(rtb_Sum4_g > 1.0E+8)) {
    /* Product: '<S90>/delta fall limit' incorporates:
     *  SampleTimeMath: '<S90>/sample time'
     *
     * About '<S90>/sample time':
     *  y = K where K = ( w * Ts )
     */
    rtb_Sum5_iu = rtb_Switch9_k * 0.01;

    /* Switch: '<S94>/Switch' incorporates:
     *  RelationalOperator: '<S94>/UpperRelop'
     */
    if (rtb_Sum4_g < rtb_Sum5_iu) {
      rtb_Sum_c = rtb_Sum5_iu;
    } else {
      rtb_Sum_c = rtb_Sum4_g;
    }

    /* End of Switch: '<S94>/Switch' */
  }

  /* End of Switch: '<S94>/Switch2' */

  /* Sum: '<S90>/Difference Inputs2' incorporates:
   *  Delay: '<S90>/Delay'
   */
  rtb_Sum4_g = rtb_Sum_c + Gen2_ref_DWork->Delay_DSTATE_j;

  /* Switch: '<S78>/Switch1' */
  if (rtb_LogicalOperator2_p1) {
    /* Switch: '<S78>/Switch3' */
    if (Gen2_ref_B->BusInput3.traj.bRateLimRejStepSizeDep) {
      rtb_Sum_c = rtb_p2HP;
    } else {
      rtb_Sum_c = rtb_Sum4_g;
    }

    /* End of Switch: '<S78>/Switch3' */
  } else {
    rtb_Sum_c = rtb_p1LP;
  }

  /* End of Switch: '<S78>/Switch1' */

  /* MinMax: '<S78>/MinMax2' */
  if ((!(rtb_Sum_c >= rtb_p1LP)) && (!rtIsNaN(rtb_p1LP))) {
    rtb_Sum_c = rtb_p1LP;
  }

  /* End of MinMax: '<S78>/MinMax2' */

  /* Sum: '<S52>/Sum11' incorporates:
   *  DiscreteIntegrator: '<S62>/Discrete-Time Integrator'
   *  Gain: '<S52>/Gain'
   */
  rtb_Sum11 = 0.0 * Gen2_ref_DWork->DiscreteTimeIntegrator_DSTATE_a + rtb_Sum_c;

  /* Product: '<S87>/delta rise limit' incorporates:
   *  Constant: '<S78>/Constant3'
   *  SampleTimeMath: '<S87>/sample time'
   *
   * About '<S87>/sample time':
   *  y = K where K = ( w * Ts )
   */
  rtb_Sum1_dh = 1.0E+8;

  /* Delay: '<S87>/Delay' incorporates:
   *  Delay: '<S78>/Variable Integer Delay'
   */
  Gen2_ref_DWork->icLoad_evr = ((((Gen2_ref_PrevZCSigState->Delay_Reset_ZCE_i ==
    1) != (int32_T)rtb_LogicalOperator1_a0) &&
    (Gen2_ref_PrevZCSigState->Delay_Reset_ZCE_i != 3)) ||
    rtb_LogicalOperator1_a0 || Gen2_ref_DWork->icLoad_evr);
  Gen2_ref_PrevZCSigState->Delay_Reset_ZCE_i = rtb_LogicalOperator1_a0;
  if (Gen2_ref_DWork->icLoad_evr) {
    Gen2_ref_DWork->Delay_DSTATE_m = rtb_p1HP;
  }

  /* Sum: '<S87>/Difference Inputs1' incorporates:
   *  Delay: '<S87>/Delay'
   *  Switch: '<S87>/etaVolConst'
   */
  rtb_Sum5_iu = rtb_p1HP - Gen2_ref_DWork->Delay_DSTATE_m;

  /* Switch: '<S91>/Switch2' incorporates:
   *  RelationalOperator: '<S91>/LowerRelop1'
   */
  if (!(rtb_Sum5_iu > 1.0E+8)) {
    /* Product: '<S87>/delta fall limit' incorporates:
     *  SampleTimeMath: '<S87>/sample time'
     *
     * About '<S87>/sample time':
     *  y = K where K = ( w * Ts )
     */
    rtb_Sum3_o = rtb_MinMax_mf * 0.01;

    /* Switch: '<S91>/Switch' incorporates:
     *  RelationalOperator: '<S91>/UpperRelop'
     */
    if (rtb_Sum5_iu < rtb_Sum3_o) {
      rtb_Sum1_dh = rtb_Sum3_o;
    } else {
      rtb_Sum1_dh = rtb_Sum5_iu;
    }

    /* End of Switch: '<S91>/Switch' */
  }

  /* End of Switch: '<S91>/Switch2' */

  /* Sum: '<S87>/Difference Inputs2' incorporates:
   *  Delay: '<S87>/Delay'
   */
  rtb_Sum5_iu = rtb_Sum1_dh + Gen2_ref_DWork->Delay_DSTATE_m;

  /* Product: '<S89>/delta rise limit' incorporates:
   *  Constant: '<S78>/Constant4'
   *  SampleTimeMath: '<S89>/sample time'
   *
   * About '<S89>/sample time':
   *  y = K where K = ( w * Ts )
   */
  rtb_Sum1_dh = 1.0E+8;

  /* Delay: '<S89>/Delay' incorporates:
   *  Delay: '<S78>/Variable Integer Delay'
   */
  Gen2_ref_DWork->icLoad_fg = ((((Gen2_ref_PrevZCSigState->Delay_Reset_ZCE_mu ==
    1) != (int32_T)rtb_LogicalOperator1_a0) &&
    (Gen2_ref_PrevZCSigState->Delay_Reset_ZCE_mu != 3)) ||
    rtb_LogicalOperator1_a0 || Gen2_ref_DWork->icLoad_fg);
  Gen2_ref_PrevZCSigState->Delay_Reset_ZCE_mu = rtb_LogicalOperator1_a0;
  if (Gen2_ref_DWork->icLoad_fg) {
    Gen2_ref_DWork->Delay_DSTATE_d = rtb_p1HP;
  }

  /* Sum: '<S89>/Difference Inputs1' incorporates:
   *  Delay: '<S89>/Delay'
   *  Switch: '<S89>/etaVolConst'
   */
  rtb_Sum3_o = rtb_p1HP - Gen2_ref_DWork->Delay_DSTATE_d;

  /* Switch: '<S93>/Switch2' incorporates:
   *  RelationalOperator: '<S93>/LowerRelop1'
   */
  if (!(rtb_Sum3_o > 1.0E+8)) {
    /* Product: '<S89>/delta fall limit' incorporates:
     *  SampleTimeMath: '<S89>/sample time'
     *
     * About '<S89>/sample time':
     *  y = K where K = ( w * Ts )
     */
    rtb_Switch9_k *= 0.01;

    /* Switch: '<S93>/Switch' incorporates:
     *  RelationalOperator: '<S93>/UpperRelop'
     */
    if (rtb_Sum3_o < rtb_Switch9_k) {
      rtb_Sum1_dh = rtb_Switch9_k;
    } else {
      rtb_Sum1_dh = rtb_Sum3_o;
    }

    /* End of Switch: '<S93>/Switch' */
  }

  /* End of Switch: '<S93>/Switch2' */

  /* Sum: '<S89>/Difference Inputs2' incorporates:
   *  Delay: '<S89>/Delay'
   */
  rtb_Switch9_k = rtb_Sum1_dh + Gen2_ref_DWork->Delay_DSTATE_d;

  /* Switch: '<S78>/Switch' */
  if (rtb_LogicalOperator2_p1) {
    /* Switch: '<S78>/Switch2' */
    if (Gen2_ref_B->BusInput3.traj.bRateLimRejStepSizeDep) {
      rtb_Sum1_dh = rtb_Sum5_iu;
    } else {
      rtb_Sum1_dh = rtb_Switch9_k;
    }

    /* End of Switch: '<S78>/Switch2' */
  } else {
    rtb_Sum1_dh = rtb_p1HP;
  }

  /* End of Switch: '<S78>/Switch' */

  /* MinMax: '<S78>/MinMax1' */
  if ((rtb_p1HP >= rtb_Sum1_dh) || rtIsNaN(rtb_Sum1_dh)) {
    rtb_MinMax1_h = rtb_p1HP;
  } else {
    rtb_MinMax1_h = rtb_Sum1_dh;
  }

  /* End of MinMax: '<S78>/MinMax1' */

  /* Product: '<S80>/delta rise limit' incorporates:
   *  Constant: '<S77>/Constant1'
   *  SampleTimeMath: '<S80>/sample time'
   *
   * About '<S80>/sample time':
   *  y = K where K = ( w * Ts )
   */
  rtb_Sum1_dh = 1.0E+8;

  /* Switch: '<S52>/Switch' */
  if (Gen2_ref_B->BusInput3.traj.bCBVrefFFonly) {
    rtb_Sum3_o = rtb_p1HP;
  } else {
    rtb_Sum3_o = rtb_p1LP;
  }

  /* End of Switch: '<S52>/Switch' */

  /* Logic: '<S77>/Logical Operator' incorporates:
   *  RelationalOperator: '<S77>/Relational Operator'
   */
  rtb_LogicalOperator2_p1 = (Gen2_ref_B->BusInput3.traj.bRateLimRejCBV &&
    (Gen2_ref_B->BusInput3.traj.rNmaxRateLimRejON > rtb_DataTypeConversion15));

  /* Logic: '<S77>/Logical Operator1' incorporates:
   *  Logic: '<S77>/Logical Operator2'
   */
  rtb_LogicalOperator1_a0 = ((!rtb_LogicalOperator2_p1) ||
    rtb_LogicalOperator2_dc);

  /* Gain: '<S77>/Gain' */
  rtb_Gain_i = 100.0 * Gen2_ref_B->BusInput3.traj.rTi_RateLimRejCBV;

  /* Delay: '<S77>/Variable Integer Delay' */
  Gen2_ref_DWork->icLoad_c =
    ((((Gen2_ref_PrevZCSigState->VariableIntegerDelay_Reset_ZC_o == 1) !=
       (int32_T)rtb_LogicalOperator1_a0) &&
      (Gen2_ref_PrevZCSigState->VariableIntegerDelay_Reset_ZC_o != 3)) ||
     rtb_LogicalOperator1_a0 || Gen2_ref_DWork->icLoad_c);
  Gen2_ref_PrevZCSigState->VariableIntegerDelay_Reset_ZC_o =
    rtb_LogicalOperator1_a0;
  if (Gen2_ref_DWork->icLoad_c) {
    for (i = 0; i < 300; i++) {
      Gen2_ref_DWork->VariableIntegerDelay_DSTATE_e[i] = rtb_p1HP;
    }
  }

  if ((rtb_Gain_i < 1.0) || rtIsNaN(rtb_Gain_i)) {
    rtb_Gain_i = rtb_p1HP;
  } else {
    if (rtb_Gain_i > 300.0) {
      i = 300;
    } else {
      delta_y = floor(rtb_Gain_i);
      if (rtIsNaN(delta_y)) {
        i = 0;
      } else {
        i = (int32_T)(uint32_T)fmod(delta_y, 4.294967296E+9);
      }
    }

    rtb_Gain_i = Gen2_ref_DWork->VariableIntegerDelay_DSTATE_e[300U - i];
  }

  /* Saturate: '<S77>/Saturation' */
  if (Gen2_ref_B->BusInput3.traj.rTi_RateLimRejCBV <= 0.01) {
    rtb_Saturation_e = 0.01;
  } else {
    rtb_Saturation_e = Gen2_ref_B->BusInput3.traj.rTi_RateLimRejCBV;
  }

  /* End of Saturate: '<S77>/Saturation' */

  /* Product: '<S77>/Divide' incorporates:
   *  Sum: '<S77>/Sum'
   */
  rtb_MinMax_a = (rtb_p1HP - rtb_Gain_i) / rtb_Saturation_e;

  /* Abs: '<S77>/Abs2' */
  rtb_Switch2_a = rtb_UkYk1_a4;

  /* Logic: '<S77>/Logical Operator3' incorporates:
   *  Gain: '<S77>/Gain3'
   *  RelationalOperator: '<S77>/Relational Operator1'
   */
  rtb_LogicalOperator3_k = (rtb_LogicalOperator1_a0 || (rtb_MinMax_a >
    -rtb_Switch2_a));

  /* Delay: '<S80>/Delay' */
  Gen2_ref_DWork->icLoad_eu = ((((Gen2_ref_PrevZCSigState->Delay_Reset_ZCE_d3 ==
    1) != (int32_T)rtb_LogicalOperator3_k) &&
    (Gen2_ref_PrevZCSigState->Delay_Reset_ZCE_d3 != 3)) ||
    rtb_LogicalOperator3_k || Gen2_ref_DWork->icLoad_eu);
  Gen2_ref_PrevZCSigState->Delay_Reset_ZCE_d3 = rtb_LogicalOperator3_k;
  if (Gen2_ref_DWork->icLoad_eu) {
    Gen2_ref_DWork->Delay_DSTATE_g2 = rtb_Sum3_o;
  }

  /* Switch: '<S80>/etaVolConst' incorporates:
   *  UnitDelay: '<S77>/Unit Delay'
   */
  if (rtb_LogicalOperator3_k) {
    rtb_UkYk1_a4 = rtb_Sum3_o;
  } else {
    rtb_UkYk1_a4 = Gen2_ref_DWork->UnitDelay_DSTATE_d;
  }

  /* End of Switch: '<S80>/etaVolConst' */

  /* Sum: '<S80>/Difference Inputs1' incorporates:
   *  Delay: '<S80>/Delay'
   */
  rtb_UkYk1_a4 -= Gen2_ref_DWork->Delay_DSTATE_g2;

  /* Abs: '<S77>/Abs' */
  rtb_Switch2_a = rtb_Switch_czo;

  /* Product: '<S77>/Divide1' incorporates:
   *  Gain: '<S77>/Gain1'
   */
  rtb_Gain_i = -rtb_Switch2_a / rtb_Saturation_e;

  /* MinMax: '<S77>/MinMax' */
  if ((rtb_MinMax_a <= rtb_Gain_i) || rtIsNaN(rtb_Gain_i)) {
    rtb_Gain_i = rtb_MinMax_a;
  }

  /* End of MinMax: '<S77>/MinMax' */

  /* Switch: '<S84>/Switch2' incorporates:
   *  RelationalOperator: '<S84>/LowerRelop1'
   */
  if (!(rtb_UkYk1_a4 > 1.0E+8)) {
    /* Product: '<S77>/Divide2' incorporates:
     *  Abs: '<S77>/Abs1'
     *  Gain: '<S77>/Gain2'
     */
    u0 = -fabs(Gen2_ref_B->BusInput3.traj.rPrDeltaMinRateLimRej) /
      rtb_Saturation_e;

    /* MinMax: '<S77>/MinMax3' */
    if ((!(u0 <= rtb_Gain_i)) && (!rtIsNaN(rtb_Gain_i))) {
      u0 = rtb_Gain_i;
    }

    /* End of MinMax: '<S77>/MinMax3' */

    /* Product: '<S80>/delta fall limit' incorporates:
     *  SampleTimeMath: '<S80>/sample time'
     *
     * About '<S80>/sample time':
     *  y = K where K = ( w * Ts )
     */
    rtb_Switch_czo = u0 * 0.01;

    /* Switch: '<S84>/Switch' incorporates:
     *  RelationalOperator: '<S84>/UpperRelop'
     */
    if (rtb_UkYk1_a4 < rtb_Switch_czo) {
      rtb_Sum1_dh = rtb_Switch_czo;
    } else {
      rtb_Sum1_dh = rtb_UkYk1_a4;
    }

    /* End of Switch: '<S84>/Switch' */
  }

  /* End of Switch: '<S84>/Switch2' */

  /* Sum: '<S80>/Difference Inputs2' incorporates:
   *  Delay: '<S80>/Delay'
   */
  rtb_Switch_czo = rtb_Sum1_dh + Gen2_ref_DWork->Delay_DSTATE_g2;

  /* Product: '<S82>/delta rise limit' incorporates:
   *  Constant: '<S77>/Constant4'
   *  SampleTimeMath: '<S82>/sample time'
   *
   * About '<S82>/sample time':
   *  y = K where K = ( w * Ts )
   */
  rtb_Sum1_dh = 1.0E+8;

  /* Delay: '<S82>/Delay' incorporates:
   *  Delay: '<S77>/Variable Integer Delay'
   */
  Gen2_ref_DWork->icLoad_ee = ((((Gen2_ref_PrevZCSigState->Delay_Reset_ZCE_c ==
    1) != (int32_T)rtb_LogicalOperator1_a0) &&
    (Gen2_ref_PrevZCSigState->Delay_Reset_ZCE_c != 3)) ||
    rtb_LogicalOperator1_a0 || Gen2_ref_DWork->icLoad_ee);
  Gen2_ref_PrevZCSigState->Delay_Reset_ZCE_c = rtb_LogicalOperator1_a0;
  if (Gen2_ref_DWork->icLoad_ee) {
    Gen2_ref_DWork->Delay_DSTATE_dm = rtb_Sum3_o;
  }

  /* Sum: '<S82>/Difference Inputs1' incorporates:
   *  Delay: '<S82>/Delay'
   *  Switch: '<S82>/etaVolConst'
   */
  rtb_UkYk1_a4 = rtb_Sum3_o - Gen2_ref_DWork->Delay_DSTATE_dm;

  /* Gain: '<S77>/Gain5' */
  rtb_MinMax_a = FILT_IN;

  /* Gain: '<S77>/Gain6' incorporates:
   *  Product: '<S77>/Divide3'
   */
  rtb_Saturation_e = -(rtb_MinMax_a / rtb_Saturation_e);

  /* Switch: '<S86>/Switch2' incorporates:
   *  RelationalOperator: '<S86>/LowerRelop1'
   */
  if (!(rtb_UkYk1_a4 > 1.0E+8)) {
    /* Product: '<S82>/delta fall limit' incorporates:
     *  SampleTimeMath: '<S82>/sample time'
     *
     * About '<S82>/sample time':
     *  y = K where K = ( w * Ts )
     */
    rtb_deltafalllimit_h0 = rtb_Saturation_e * 0.01;

    /* Switch: '<S86>/Switch' incorporates:
     *  RelationalOperator: '<S86>/UpperRelop'
     */
    if (rtb_UkYk1_a4 < rtb_deltafalllimit_h0) {
      rtb_Sum1_dh = rtb_deltafalllimit_h0;
    } else {
      rtb_Sum1_dh = rtb_UkYk1_a4;
    }

    /* End of Switch: '<S86>/Switch' */
  }

  /* End of Switch: '<S86>/Switch2' */

  /* Sum: '<S82>/Difference Inputs2' incorporates:
   *  Delay: '<S82>/Delay'
   */
  rtb_UkYk1_a4 = rtb_Sum1_dh + Gen2_ref_DWork->Delay_DSTATE_dm;

  /* Switch: '<S77>/Switch1' */
  if (rtb_LogicalOperator2_p1) {
    /* Switch: '<S77>/Switch3' */
    if (Gen2_ref_B->BusInput3.traj.bRateLimRejStepSizeDep) {
      rtb_Sum1_dh = rtb_Switch_czo;
    } else {
      rtb_Sum1_dh = rtb_UkYk1_a4;
    }

    /* End of Switch: '<S77>/Switch3' */
  } else {
    rtb_Sum1_dh = rtb_Sum3_o;
  }

  /* End of Switch: '<S77>/Switch1' */

  /* MinMax: '<S77>/MinMax2' */
  if ((!(rtb_Sum1_dh >= rtb_Sum3_o)) && (!rtIsNaN(rtb_Sum3_o))) {
    rtb_Sum1_dh = rtb_Sum3_o;
  }

  /* End of MinMax: '<S77>/MinMax2' */

  /* Sum: '<S52>/Sum7' incorporates:
   *  DiscreteIntegrator: '<S62>/Discrete-Time Integrator'
   */
  rtb_Sum7_l5 = Gen2_ref_DWork->DiscreteTimeIntegrator_DSTATE_a + rtb_Sum1_dh;

  /* Product: '<S79>/delta rise limit' incorporates:
   *  Constant: '<S77>/Constant3'
   *  SampleTimeMath: '<S79>/sample time'
   *
   * About '<S79>/sample time':
   *  y = K where K = ( w * Ts )
   */
  rtb_Sum1_dh = 1.0E+8;

  /* Delay: '<S79>/Delay' incorporates:
   *  Delay: '<S77>/Variable Integer Delay'
   */
  Gen2_ref_DWork->icLoad_ki = ((((Gen2_ref_PrevZCSigState->Delay_Reset_ZCE_p ==
    1) != (int32_T)rtb_LogicalOperator1_a0) &&
    (Gen2_ref_PrevZCSigState->Delay_Reset_ZCE_p != 3)) ||
    rtb_LogicalOperator1_a0 || Gen2_ref_DWork->icLoad_ki);
  Gen2_ref_PrevZCSigState->Delay_Reset_ZCE_p = rtb_LogicalOperator1_a0;
  if (Gen2_ref_DWork->icLoad_ki) {
    Gen2_ref_DWork->Delay_DSTATE_jl = rtb_p1HP;
  }

  /* Sum: '<S79>/Difference Inputs1' incorporates:
   *  Delay: '<S79>/Delay'
   *  Switch: '<S79>/etaVolConst'
   */
  rtb_deltafalllimit_h0 = rtb_p1HP - Gen2_ref_DWork->Delay_DSTATE_jl;

  /* Switch: '<S83>/Switch2' incorporates:
   *  RelationalOperator: '<S83>/LowerRelop1'
   */
  if (!(rtb_deltafalllimit_h0 > 1.0E+8)) {
    /* Product: '<S79>/delta fall limit' incorporates:
     *  SampleTimeMath: '<S79>/sample time'
     *
     * About '<S79>/sample time':
     *  y = K where K = ( w * Ts )
     */
    rtb_Gain_i *= 0.01;

    /* Switch: '<S83>/Switch' incorporates:
     *  RelationalOperator: '<S83>/UpperRelop'
     */
    if (rtb_deltafalllimit_h0 < rtb_Gain_i) {
      rtb_Sum1_dh = rtb_Gain_i;
    } else {
      rtb_Sum1_dh = rtb_deltafalllimit_h0;
    }

    /* End of Switch: '<S83>/Switch' */
  }

  /* End of Switch: '<S83>/Switch2' */

  /* Sum: '<S79>/Difference Inputs2' incorporates:
   *  Delay: '<S79>/Delay'
   */
  rtb_Gain_i = rtb_Sum1_dh + Gen2_ref_DWork->Delay_DSTATE_jl;

  /* Product: '<S81>/delta rise limit' incorporates:
   *  Constant: '<S77>/Constant4'
   *  SampleTimeMath: '<S81>/sample time'
   *
   * About '<S81>/sample time':
   *  y = K where K = ( w * Ts )
   */
  rtb_Sum1_dh = 1.0E+8;

  /* Delay: '<S81>/Delay' incorporates:
   *  Delay: '<S77>/Variable Integer Delay'
   */
  Gen2_ref_DWork->icLoad_h3 = ((((Gen2_ref_PrevZCSigState->Delay_Reset_ZCE_ih ==
    1) != (int32_T)rtb_LogicalOperator1_a0) &&
    (Gen2_ref_PrevZCSigState->Delay_Reset_ZCE_ih != 3)) ||
    rtb_LogicalOperator1_a0 || Gen2_ref_DWork->icLoad_h3);
  Gen2_ref_PrevZCSigState->Delay_Reset_ZCE_ih = rtb_LogicalOperator1_a0;
  if (Gen2_ref_DWork->icLoad_h3) {
    Gen2_ref_DWork->Delay_DSTATE_h = rtb_p1HP;
  }

  /* Sum: '<S81>/Difference Inputs1' incorporates:
   *  Delay: '<S81>/Delay'
   *  Switch: '<S81>/etaVolConst'
   */
  rtb_deltafalllimit_h0 = rtb_p1HP - Gen2_ref_DWork->Delay_DSTATE_h;

  /* Switch: '<S85>/Switch2' incorporates:
   *  RelationalOperator: '<S85>/LowerRelop1'
   */
  if (!(rtb_deltafalllimit_h0 > 1.0E+8)) {
    /* Product: '<S81>/delta fall limit' incorporates:
     *  SampleTimeMath: '<S81>/sample time'
     *
     * About '<S81>/sample time':
     *  y = K where K = ( w * Ts )
     */
    rtb_Saturation_e *= 0.01;
```
